    R101_3축_프론트_I_RB_PROG_ECHO_8 AT %MW84012.3 : BOOL;
    R101_3축_프론트_I_RB_SP3_8 AT %MW84013.8 : BOOL;
    R101_3축_프론트_I_RB_SP3_9 AT %MW84013.9 : BOOL;
    R101_3축_프론트_I_RB_SPARE_WORD_4 AT %MW84014 : WORD;
    R101_3축_프론트_I_RB_SP_1_12 AT %MW84011.12 : BOOL;
    R101_3축_프론트_I_RB_SP_1_13 AT %MW84011.13 : BOOL;
    R101_3축_프론트_I_RB_SP_1_14 AT %MW84011.14 : BOOL;
    R101_3축_프론트_I_RB_SP_1_15 AT %MW84011.15 : BOOL;
    R101_3축_프론트_I_RB_TC_이상 AT %MW84012.8 : BOOL;
    R101_3축_프론트_I_RB_TIP_CHANGE AT %MW84013.13 : BOOL;
    R101_3축_프론트_I_RB_TIP_DRESSING AT %MW84010.7 : BOOL;
    R101_3축_프론트_I_RB__PLT_카운터리셋완료 AT %MW84013.10 : BOOL;
    R101_3축_프론트_I_RB_공기압_이상 AT %MW84012.9 : BOOL;
    R101_3축_프론트_I_RB_냉각수_이상 AT %MW84012.10 : BOOL;
    R101_3축_프론트_I_RB_비상정지_NC AT %MW84010.8 : BOOL;
    R101_3축_프론트_I_RB_비전이상 AT %MW84012.14 : BOOL;
    R101_3축_프론트_I_RB_실러이상 AT %MW84012.13 : BOOL;
    R101_3축_프론트_I_RB_용접카운터이상 AT %MW84012.15 : BOOL;
    R101_3축_프론트_I_RB_용접타점수 AT %MW84015 : WORD;
    R101_3축_프론트_I_RB_운전준비 AT %MW84010.3 : BOOL;
    R101_3축_프론트_I_RB_원위치 AT %MW84010.0 : BOOL;
    R101_3축_프론트_I_RB_이상리셋 AT %MW84010.2 : BOOL;
    R101_3축_프론트_I_RB_자동 AT %MW84010.4 : BOOL;
    R101_3축_프론트_I_RB_자동기동 AT %MW84010.5 : BOOL;
    R101_3축_프론트_I_RB_최종_작업완료 AT %MW84010.1 : BOOL;
    R101_3축_프론트_I_RB_통신이상 AT %MW84012.12 : BOOL;
    R101_3축_프론트_M_I_RB_1차_작업완료 AT %MW20011.2 : BOOL;
    R101_3축_프론트_M_I_RB_2차_작업완료 AT %MW20011.3 : BOOL;
    R101_3축_프론트_M_I_RB_3차_작업완료 AT %MW20011.4 : BOOL;
    R101_3축_프론트_M_I_RB_4차_작업완료 AT %MW20011.5 : BOOL;
    R101_3축_프론트_M_I_RB_5차_작업완료 AT %MW20011.6 : BOOL;
    R101_3축_프론트_M_I_RB_6차_작업완료 AT %MW20011.7 : BOOL;
    R101_3축_프론트_M_I_RB_7차_작업완료 AT %MW20011.8 : BOOL;
    R101_3축_프론트_M_I_RB_PAUSE_보조 AT %MW20010.5 : BOOL;
    R101_3축_프론트_M_I_RB_PLC_RUN_CHK_이상 AT %MW20010.7 : BOOL;
    R101_3축_프론트_M_I_RB_간섭무_1 AT %MW20012.0 : BOOL;
    R101_3축_프론트_M_I_RB_간섭무_10 AT %MW20012.9 : BOOL;
    R101_3축_프론트_M_I_RB_간섭무_11 AT %MW20012.10 : BOOL;
    R101_3축_프론트_M_I_RB_간섭무_12 AT %MW20012.11 : BOOL;
    R101_3축_프론트_M_I_RB_간섭무_2 AT %MW20012.1 : BOOL;
    R101_3축_프론트_M_I_RB_간섭무_3 AT %MW20012.2 : BOOL;
    R101_3축_프론트_M_I_RB_간섭무_4 AT %MW20012.3 : BOOL;
    R101_3축_프론트_M_I_RB_간섭무_5 AT %MW20012.4 : BOOL;
    R101_3축_프론트_M_I_RB_간섭무_6 AT %MW20012.5 : BOOL;
    R101_3축_프론트_M_I_RB_간섭무_7 AT %MW20012.6 : BOOL;
    R101_3축_프론트_M_I_RB_간섭무_8 AT %MW20012.7 : BOOL;
    R101_3축_프론트_M_I_RB_간섭무_9 AT %MW20012.8 : BOOL;
    R101_3축_프론트_M_I_RB_비상정지 AT %MW20010.4 : BOOL;
    R101_3축_프론트_M_I_RB_운전준비 AT %MW20010.0 : BOOL;
    R101_3축_프론트_M_I_RB_원위치 AT %MW20010.3 : BOOL;
    R101_3축_프론트_M_I_RB_이상 AT %MW20010.2 : BOOL;
    R101_3축_프론트_M_I_RB_자동 AT %MW20010.1 : BOOL;
    R101_3축_프론트_M_I_RB_최종작업완료 AT %MW20011.0 : BOOL;
    R101_3축_프론트_M_I_RB_프로그램_이상 AT %MW20010.6 : BOOL;
    R101_3축_프론트_M_O_RB_1_CYCLE_SET AT %MW21010.3 : BOOL;
    R101_3축_프론트_M_O_RB_1_CYCLE_리셋 AT %MW21010.4 : BOOL;
    R101_3축_프론트_M_O_RB_1차_작업완료_리셋 AT %MW21012.0 : BOOL;
    R101_3축_프론트_M_O_RB_2차_작업완료_리셋 AT %MW21012.1 : BOOL;
    R101_3축_프론트_M_O_RB_2차_진입OK AT %MW21011.8 : BOOL;
    R101_3축_프론트_M_O_RB_3차_작업완료_리셋 AT %MW21012.2 : BOOL;
    R101_3축_프론트_M_O_RB_3차_진입OK AT %MW21011.9 : BOOL;
    R101_3축_프론트_M_O_RB_4차_작업완료_리셋 AT %MW21012.3 : BOOL;
    R101_3축_프론트_M_O_RB_4차_진입OK AT %MW21011.10 : BOOL;
    R101_3축_프론트_M_O_RB_5차_작업완료_리셋 AT %MW21012.4 : BOOL;
    R101_3축_프론트_M_O_RB_5차_진입OK AT %MW21011.11 : BOOL;
    R101_3축_프론트_M_O_RB_6차_작업완료_리셋 AT %MW21012.5 : BOOL;
    R101_3축_프론트_M_O_RB_6차_진입OK AT %MW21011.12 : BOOL;
    R101_3축_프론트_M_O_RB_7차_작업완료_리셋 AT %MW21012.6 : BOOL;
    R101_3축_프론트_M_O_RB_7차_진입OK AT %MW21011.13 : BOOL;
    R101_3축_프론트_M_O_RB_ATD_OK AT %MW21010.6 : BOOL;
    R101_3축_프론트_M_O_RB_PLT_10_진입OK AT %MW21013.10 : BOOL;
    R101_3축_프론트_M_O_RB_PLT_11_진입OK AT %MW21013.11 : BOOL;
    R101_3축_프론트_M_O_RB_PLT_12_진입OK AT %MW21013.12 : BOOL;
    R101_3축_프론트_M_O_RB_PLT_1_진입OK AT %MW21013.1 : BOOL;
    R101_3축_프론트_M_O_RB_PLT_2_진입OK AT %MW21013.2 : BOOL;
    R101_3축_프론트_M_O_RB_PLT_3_진입OK AT %MW21013.3 : BOOL;
    R101_3축_프론트_M_O_RB_PLT_4_진입OK AT %MW21013.4 : BOOL;
    R101_3축_프론트_M_O_RB_PLT_5_진입OK AT %MW21013.5 : BOOL;
    R101_3축_프론트_M_O_RB_PLT_6_진입OK AT %MW21013.6 : BOOL;
    R101_3축_프론트_M_O_RB_PLT_7_진입OK AT %MW21013.7 : BOOL;
    R101_3축_프론트_M_O_RB_PLT_8_진입OK AT %MW21013.8 : BOOL;
    R101_3축_프론트_M_O_RB_PLT_9_진입OK AT %MW21013.9 : BOOL;
    R101_3축_프론트_M_O_RB_PLT_카운터리셋_보조 AT %MW21010.10 : BOOL;
    R101_3축_프론트_M_O_RB_RESTART_OK AT %MW21010.2 : BOOL;
    R101_3축_프론트_M_O_RB_START_OK AT %MW21010.0 : BOOL;
    R101_3축_프론트_M_O_RB_TEST_MODE_5000회 AT %MW21010.12 : BOOL;
    R101_3축_프론트_M_O_RB_TIP_교체_시작 AT %MW21010.7 : BOOL;
    R101_3축_프론트_M_O_RB_TIP_교체_완료 AT %MW21010.8 : BOOL;
    R101_3축_프론트_M_O_RB_VIP_MODE AT %MW21010.11 : BOOL;
    R101_3축_프론트_M_O_RB_냉각수_차단_요청 AT %MW21010.9 : BOOL;
    R101_3축_프론트_M_O_RB_진입OK_AX차종 AT %MW21011.0 : BOOL;
    R101_3축_프론트_M_O_RB_진입OK_B차종 AT %MW21011.1 : BOOL;
    R101_3축_프론트_M_O_RB_진입OK_C차종 AT %MW21011.2 : BOOL;
    R101_3축_프론트_M_O_RB_진입OK_D차종 AT %MW21011.3 : BOOL;
    R101_3축_프론트_M_O_RB_진입OK_E차종 AT %MW21011.4 : BOOL;
    R101_3축_프론트_M_O_RB_진입OK_F차종 AT %MW21011.5 : BOOL;
    R101_3축_프론트_M_O_RB_진입OK_G차종 AT %MW21011.6 : BOOL;
    R101_3축_프론트_M_O_RB_진입OK_H차종 AT %MW21011.7 : BOOL;
    R101_3축_프론트_M_O_RB_최종_작업완료_리셋 AT %MW21010.5 : BOOL;
    R101_3축_프론트_M_O_RB_프로그램_OK AT %MW21010.1 : BOOL;
    R101_3축_프론트_M_RB_PROG_NO AT %MW20014 : WORD;
    R101_3축_프론트_O_RB_0_5S_통신_CHK AT %MW94013.14 : BOOL;
    R101_3축_프론트_O_RB_2차_진입OK AT %MW94011.8 : BOOL;
    R101_3축_프론트_O_RB_3차_진입OK AT %MW94011.9 : BOOL;
    R101_3축_프론트_O_RB_4차_진입OK AT %MW94011.10 : BOOL;
    R101_3축_프론트_O_RB_5차_진입OK AT %MW94011.11 : BOOL;
    R101_3축_프론트_O_RB_6차_진입OK AT %MW94011.12 : BOOL;
    R101_3축_프론트_O_RB_7차_진입OK AT %MW94011.13 : BOOL;
    R101_3축_프론트_O_RB_AX_1차_진입OK AT %MW94011.0 : BOOL;
    R101_3축_프론트_O_RB_B_1차_진입OK AT %MW94011.1 : BOOL;
    R101_3축_프론트_O_RB_C_1차_진입OK AT %MW94011.2 : BOOL;
    R101_3축_프론트_O_RB_D_1차_진입OK AT %MW94011.3 : BOOL;
    R101_3축_프론트_O_RB_EACH_작업완료_리셋 AT %MW94010.14 : BOOL;
    R101_3축_프론트_O_RB_EXT_READY AT %MW94010.11 : BOOL;
    R101_3축_프론트_O_RB_E_1차_진입OK AT %MW94011.4 : BOOL;
    R101_3축_프론트_O_RB_F_1차_진입OK AT %MW94011.5 : BOOL;
    R101_3축_프론트_O_RB_GATE_OPEN_NC AT %MW94013.11 : BOOL;
    R101_3축_프론트_O_RB_G_1차_진입OK AT %MW94011.6 : BOOL;
    R101_3축_프론트_O_RB_H_1차_진입OK AT %MW94011.7 : BOOL;
    R101_3축_프론트_O_RB_MUTUAL_INT1 AT %MW94013.0 : BOOL;
    R101_3축_프론트_O_RB_MUTUAL_INT2 AT %MW94013.1 : BOOL;
    R101_3축_프론트_O_RB_MUTUAL_INT3 AT %MW94013.2 : BOOL;
    R101_3축_프론트_O_RB_MUTUAL_INT4 AT %MW94013.3 : BOOL;
    R101_3축_프론트_O_RB_MUTUAL_INT5 AT %MW94013.4 : BOOL;
    R101_3축_프론트_O_RB_MUTUAL_INT6 AT %MW94013.5 : BOOL;
    R101_3축_프론트_O_RB_MUTUAL_INT7 AT %MW94013.6 : BOOL;
    R101_3축_프론트_O_RB_MUTUAL_INT8 AT %MW94013.7 : BOOL;
    R101_3축_프론트_O_RB_OUTPUT AT %MW94010 : ARRAY[0..3] OF WORD;
    R101_3축_프론트_O_RB_PAUSE_NC AT %MW94010.13 : BOOL;
    R101_3축_프론트_O_RB_PLT10_진입OK AT %MW94012.9 : BOOL;
    R101_3축_프론트_O_RB_PLT11_진입OK AT %MW94012.10 : BOOL;
    R101_3축_프론트_O_RB_PLT12_진입OK AT %MW94012.11 : BOOL;
    R101_3축_프론트_O_RB_PLT1_진입OK AT %MW94012.0 : BOOL;
    R101_3축_프론트_O_RB_PLT2_진입OK AT %MW94012.1 : BOOL;
    R101_3축_프론트_O_RB_PLT3_진입OK AT %MW94012.2 : BOOL;
    R101_3축_프론트_O_RB_PLT4_진입OK AT %MW94012.3 : BOOL;
    R101_3축_프론트_O_RB_PLT5_진입OK AT %MW94012.4 : BOOL;
    R101_3축_프론트_O_RB_PLT6_진입OK AT %MW94012.5 : BOOL;
    R101_3축_프론트_O_RB_PLT7_진입OK AT %MW94012.6 : BOOL;
    R101_3축_프론트_O_RB_PLT8_진입OK AT %MW94012.7 : BOOL;
    R101_3축_프론트_O_RB_PLT9_진입OK AT %MW94012.8 : BOOL;
    R101_3축_프론트_O_RB_PLT_COUNT_리셋_COND AT %MW94013.10 : BOOL;
    R101_3축_프론트_O_RB_PROG_선택1 AT %MW94010.0 : BOOL;
    R101_3축_프론트_O_RB_PROG_선택128 AT %MW94010.7 : BOOL;
    R101_3축_프론트_O_RB_PROG_선택16 AT %MW94010.4 : BOOL;
    R101_3축_프론트_O_RB_PROG_선택2 AT %MW94010.1 : BOOL;
    R101_3축_프론트_O_RB_PROG_선택32 AT %MW94010.5 : BOOL;
    R101_3축_프론트_O_RB_PROG_선택4 AT %MW94010.2 : BOOL;
    R101_3축_프론트_O_RB_PROG_선택64 AT %MW94010.6 : BOOL;
    R101_3축_프론트_O_RB_PROG_선택8 AT %MW94010.3 : BOOL;
    R101_3축_프론트_O_RB_SP_1_14 AT %MW94011.14 : BOOL;
    R101_3축_프론트_O_RB_SP_1_15 AT %MW94011.15 : BOOL;
    R101_3축_프론트_O_RB_SP_2_12 AT %MW94012.12 : BOOL;
    R101_3축_프론트_O_RB_SP_2_13 AT %MW94012.13 : BOOL;
    R101_3축_프론트_O_RB_SP_2_14 AT %MW94012.14 : BOOL;
    R101_3축_프론트_O_RB_SP_5000TH_ON AT %MW94012.15 : BOOL;
    R101_3축_프론트_O_RB_TIP_CHANGE_END AT %MW94013.9 : BOOL;
    R101_3축_프론트_O_RB_TIP_CHANGE_START AT %MW94013.8 : BOOL;
    R101_3축_프론트_O_RB_TIP_DRESS_SATRT AT %MW94010.12 : BOOL;
    R101_3축_프론트_O_RB_VIP_MODE AT %MW94013.15 : BOOL;
    R101_3축_프론트_O_RB_기동 AT %MW94010.9 : BOOL;
    R101_3축_프론트_O_RB_냉각수차단 AT %MW94010.15 : BOOL;
    R101_3축_프론트_O_RB_부저정지 AT %MW94013.13 : BOOL;
    R101_3축_프론트_O_RB_비상정지_NC AT %MW94013.12 : BOOL;
    R101_3축_프론트_O_RB_이상_리셋 AT %MW94010.10 : BOOL;
    R101_3축_프론트_O_RB_작업완료_리셋 AT %MW94010.8 : BOOL;
    R102_1_1_I_RB_0_5_COMM_CHK AT %MW84093.14 : BOOL;
    R102_1_1_I_RB_10차_간섭무 AT %MW84091.9 : BOOL;
    R102_1_1_I_RB_11차_간섭무 AT %MW84091.10 : BOOL;
    R102_1_1_I_RB_12차_간섭무 AT %MW84091.11 : BOOL;
    R102_1_1_I_RB_1차_간섭무 AT %MW84091.0 : BOOL;
    R102_1_1_I_RB_1차_작업완료 AT %MW84090.9 : BOOL;
    R102_1_1_I_RB_2차_간섭무 AT %MW84091.1 : BOOL;
    R102_1_1_I_RB_2차_작업완료 AT %MW84090.10 : BOOL;
    R102_1_1_I_RB_3차_간섭무 AT %MW84091.2 : BOOL;
    R102_1_1_I_RB_3차_작업완료 AT %MW84090.11 : BOOL;
    R102_1_1_I_RB_4차_간섭무 AT %MW84091.3 : BOOL;
    R102_1_1_I_RB_4차_작업완료 AT %MW84090.12 : BOOL;
    R102_1_1_I_RB_5차_간섭무 AT %MW84091.4 : BOOL;
    R102_1_1_I_RB_5차_작업완료 AT %MW84090.13 : BOOL;
    R102_1_1_I_RB_6차_간섭무 AT %MW84091.5 : BOOL;
    R102_1_1_I_RB_6차_작업완료 AT %MW84090.14 : BOOL;
    R102_1_1_I_RB_7차_간섭무 AT %MW84091.6 : BOOL;
    R102_1_1_I_RB_7차_작업완료 AT %MW84090.15 : BOOL;
    R102_1_1_I_RB_8차_간섭무 AT %MW84091.7 : BOOL;
    R102_1_1_I_RB_9차_간섭무 AT %MW84091.8 : BOOL;
    R102_1_1_I_RB_AB_NORMAL_선택 AT %MW84090.6 : BOOL;
    R102_1_1_I_RB_GUN1_FIXED_TIP AT %MW84097 : WORD;
    R102_1_1_I_RB_GUN1_MOVING_TIP AT %MW84096 : WORD;
    R102_1_1_I_RB_GUN2_FIXED_TIP AT %MW84099 : WORD;
    R102_1_1_I_RB_GUN2_MOVING_TIP AT %MW84098 : WORD;
    R102_1_1_I_RB_INPUT AT %MW84090 : ARRAY[0..3] OF WORD;
    R102_1_1_I_RB_LS_이상 AT %MW84092.11 : BOOL;
    R102_1_1_I_RB_MOTOR_MC_ON AT %MW84093.15 : BOOL;
    R102_1_1_I_RB_MUTUAL_INT1 AT %MW84093.0 : BOOL;
    R102_1_1_I_RB_MUTUAL_INT2 AT %MW84093.1 : BOOL;
    R102_1_1_I_RB_MUTUAL_INT3 AT %MW84093.2 : BOOL;
    R102_1_1_I_RB_MUTUAL_INT4 AT %MW84093.3 : BOOL;
    R102_1_1_I_RB_MUTUAL_INT5 AT %MW84093.4 : BOOL;
    R102_1_1_I_RB_MUTUAL_INT6 AT %MW84093.5 : BOOL;
    R102_1_1_I_RB_MUTUAL_INT7 AT %MW84093.6 : BOOL;
    R102_1_1_I_RB_MUTUAL_INT8 AT %MW84093.7 : BOOL;
    R102_1_1_I_RB_PLT_UNLOAD_완료 AT %MW84093.11 : BOOL;
    R102_1_1_I_RB_PLT_최종UNLOAD_완료 AT %MW84093.12 : BOOL;
    R102_1_1_I_RB_PROG_ECHO_1 AT %MW84092.0 : BOOL;
    R102_1_1_I_RB_PROG_ECHO_128 AT %MW84092.7 : BOOL;
    R102_1_1_I_RB_PROG_ECHO_16 AT %MW84092.4 : BOOL;
    R102_1_1_I_RB_PROG_ECHO_2 AT %MW84092.1 : BOOL;
    R102_1_1_I_RB_PROG_ECHO_32 AT %MW84092.5 : BOOL;
    R102_1_1_I_RB_PROG_ECHO_4 AT %MW84092.2 : BOOL;
    R102_1_1_I_RB_PROG_ECHO_64 AT %MW84092.6 : BOOL;
    R102_1_1_I_RB_PROG_ECHO_8 AT %MW84092.3 : BOOL;
    R102_1_1_I_RB_SP3_8 AT %MW84093.8 : BOOL;
    R102_1_1_I_RB_SP3_9 AT %MW84093.9 : BOOL;
    R102_1_1_I_RB_SPARE_WORD_4 AT %MW84094 : WORD;
    R102_1_1_I_RB_SP_1_12 AT %MW84091.12 : BOOL;
    R102_1_1_I_RB_SP_1_13 AT %MW84091.13 : BOOL;
    R102_1_1_I_RB_SP_1_14 AT %MW84091.14 : BOOL;
    R102_1_1_I_RB_SP_1_15 AT %MW84091.15 : BOOL;
    R102_1_1_I_RB_TC_이상 AT %MW84092.8 : BOOL;
    R102_1_1_I_RB_TIP_CHANGE AT %MW84093.13 : BOOL;
    R102_1_1_I_RB_TIP_DRESSING AT %MW84090.7 : BOOL;
    R102_1_1_I_RB__PLT_카운터리셋완료 AT %MW84093.10 : BOOL;
    R102_1_1_I_RB_공기압_이상 AT %MW84092.9 : BOOL;
    R102_1_1_I_RB_냉각수_이상 AT %MW84092.10 : BOOL;
    R102_1_1_I_RB_비상정지_NC AT %MW84090.8 : BOOL;
    R102_1_1_I_RB_비전이상 AT %MW84092.14 : BOOL;
    R102_1_1_I_RB_실러이상 AT %MW84092.13 : BOOL;
    R102_1_1_I_RB_용접카운터이상 AT %MW84092.15 : BOOL;
    R102_1_1_I_RB_용접타점수 AT %MW84095 : WORD;
    R102_1_1_I_RB_운전준비 AT %MW84090.3 : BOOL;
    R102_1_1_I_RB_원위치 AT %MW84090.0 : BOOL;
    R102_1_1_I_RB_이상리셋 AT %MW84090.2 : BOOL;
    R102_1_1_I_RB_자동 AT %MW84090.4 : BOOL;
    R102_1_1_I_RB_자동기동 AT %MW84090.5 : BOOL;
    R102_1_1_I_RB_최종_작업완료 AT %MW84090.1 : BOOL;
    R102_1_1_I_RB_통신이상 AT %MW84092.12 : BOOL;
    R102_1_1_M_DATA_삭제_PLS AT %MW9002.0 : BOOL; (* R102_1_1_M_DATA_삭제_PLS *)
    R102_1_1_M_DATA_삭제_SIGN AT %MW9002.1 : BOOL; (* R102_1_1_M_DATA_삭제_SIGN *)
    R102_1_1_M_DATA_삭제_완료 AT %MW9002.2 : BOOL; (* R102_1_1_M_DATA_삭제_완료 *)
    R102_1_1_M_DATA_전송_MEMO AT %MW9002.8 : BOOL; (* R102_1_1_M_DATA_전송_MEMO *)
    R102_1_1_M_DATA_전송_PLS AT %MW9002.9 : BOOL; (* R102_1_1_M_DATA_전송_PLS *)
    R102_1_1_M_DATA_전송_SIGN AT %MW9002.10 : BOOL; (* R102_1_1_M_DATA_전송_SIGN *)
    R102_1_1_M_DATA_전송_완료 AT %MW9002.11 : BOOL; (* R102_1_1_M_DATA_전송_완료 *)
    R102_1_1_M_I_RB_1차_작업완료 AT %MW20091.2 : BOOL;
    R102_1_1_M_I_RB_2차_작업완료 AT %MW20091.3 : BOOL;
    R102_1_1_M_I_RB_3차_작업완료 AT %MW20091.4 : BOOL;
    R102_1_1_M_I_RB_4차_작업완료 AT %MW20091.5 : BOOL;
    R102_1_1_M_I_RB_5차_작업완료 AT %MW20091.6 : BOOL;
    R102_1_1_M_I_RB_6차_작업완료 AT %MW20091.7 : BOOL;
    R102_1_1_M_I_RB_7차_작업완료 AT %MW20091.8 : BOOL;
    R102_1_1_M_I_RB_PAUSE_보조 AT %MW20090.5 : BOOL;
    R102_1_1_M_I_RB_PLC_RUN_CHK_이상 AT %MW20090.7 : BOOL;
    R102_1_1_M_I_RB_간섭무_1 AT %MW20092.0 : BOOL;
    R102_1_1_M_I_RB_간섭무_10 AT %MW20092.9 : BOOL;
    R102_1_1_M_I_RB_간섭무_11 AT %MW20092.10 : BOOL;
    R102_1_1_M_I_RB_간섭무_12 AT %MW20092.11 : BOOL;
    R102_1_1_M_I_RB_간섭무_2 AT %MW20092.1 : BOOL;
    R102_1_1_M_I_RB_간섭무_3 AT %MW20092.2 : BOOL;
    R102_1_1_M_I_RB_간섭무_4 AT %MW20092.3 : BOOL;
    R102_1_1_M_I_RB_간섭무_5 AT %MW20092.4 : BOOL;
    R102_1_1_M_I_RB_간섭무_6 AT %MW20092.5 : BOOL;
    R102_1_1_M_I_RB_간섭무_7 AT %MW20092.6 : BOOL;
    R102_1_1_M_I_RB_간섭무_8 AT %MW20092.7 : BOOL;
    R102_1_1_M_I_RB_간섭무_9 AT %MW20092.8 : BOOL;
    R102_1_1_M_I_RB_비상정지 AT %MW20090.4 : BOOL;
    R102_1_1_M_I_RB_운전준비 AT %MW20090.0 : BOOL;
    R102_1_1_M_I_RB_원위치 AT %MW20090.3 : BOOL;
    R102_1_1_M_I_RB_이상 AT %MW20090.2 : BOOL;
    R102_1_1_M_I_RB_자동 AT %MW20090.1 : BOOL;
    R102_1_1_M_I_RB_최종작업완료 AT %MW20091.0 : BOOL;
    R102_1_1_M_I_RB_프로그램_이상 AT %MW20090.6 : BOOL;
    R102_1_1_M_O_RB_1_CYCLE_SET AT %MW21090.3 : BOOL;
    R102_1_1_M_O_RB_1_CYCLE_리셋 AT %MW21090.4 : BOOL;
    R102_1_1_M_O_RB_1차_작업완료_리셋 AT %MW21092.0 : BOOL;
    R102_1_1_M_O_RB_2차_작업완료_리셋 AT %MW21092.1 : BOOL;
    R102_1_1_M_O_RB_2차_진입OK AT %MW21091.8 : BOOL;
    R102_1_1_M_O_RB_3차_작업완료_리셋 AT %MW21092.2 : BOOL;
    R102_1_1_M_O_RB_3차_진입OK AT %MW21091.9 : BOOL;
    R102_1_1_M_O_RB_4차_작업완료_리셋 AT %MW21092.3 : BOOL;
    R102_1_1_M_O_RB_4차_진입OK AT %MW21091.10 : BOOL;
    R102_1_1_M_O_RB_5차_작업완료_리셋 AT %MW21092.4 : BOOL;
    R102_1_1_M_O_RB_5차_진입OK AT %MW21091.11 : BOOL;
    R102_1_1_M_O_RB_6차_작업완료_리셋 AT %MW21092.5 : BOOL;
    R102_1_1_M_O_RB_6차_진입OK AT %MW21091.12 : BOOL;
    R102_1_1_M_O_RB_7차_작업완료_리셋 AT %MW21092.6 : BOOL;
    R102_1_1_M_O_RB_7차_진입OK AT %MW21091.13 : BOOL;
    R102_1_1_M_O_RB_ATD_OK AT %MW21090.6 : BOOL;
    R102_1_1_M_O_RB_PLT_10_진입OK AT %MW21093.10 : BOOL;
    R102_1_1_M_O_RB_PLT_11_진입OK AT %MW21093.11 : BOOL;
    R102_1_1_M_O_RB_PLT_12_진입OK AT %MW21093.12 : BOOL;
    R102_1_1_M_O_RB_PLT_1_진입OK AT %MW21093.1 : BOOL;
    R102_1_1_M_O_RB_PLT_2_진입OK AT %MW21093.2 : BOOL;
    R102_1_1_M_O_RB_PLT_3_진입OK AT %MW21093.3 : BOOL;
    R102_1_1_M_O_RB_PLT_4_진입OK AT %MW21093.4 : BOOL;
    R102_1_1_M_O_RB_PLT_5_진입OK AT %MW21093.5 : BOOL;
    R102_1_1_M_O_RB_PLT_6_진입OK AT %MW21093.6 : BOOL;
    R102_1_1_M_O_RB_PLT_7_진입OK AT %MW21093.7 : BOOL;
    R102_1_1_M_O_RB_PLT_8_진입OK AT %MW21093.8 : BOOL;
    R102_1_1_M_O_RB_PLT_9_진입OK AT %MW21093.9 : BOOL;
    R102_1_1_M_O_RB_PLT_카운터리셋_보조 AT %MW21090.10 : BOOL;
    R102_1_1_M_O_RB_RESTART_OK AT %MW21090.2 : BOOL;
    R102_1_1_M_O_RB_START_OK AT %MW21090.0 : BOOL;
    R102_1_1_M_O_RB_TEST_MODE_5000회 AT %MW21090.12 : BOOL;
    R102_1_1_M_O_RB_TIP_교체_시작 AT %MW21090.7 : BOOL;
    R102_1_1_M_O_RB_TIP_교체_완료 AT %MW21090.8 : BOOL;
    R102_1_1_M_O_RB_VIP_MODE AT %MW21090.11 : BOOL;
    R102_1_1_M_O_RB_냉각수_차단_요청 AT %MW21090.9 : BOOL;
    R102_1_1_M_O_RB_진입OK_AX차종 AT %MW21091.0 : BOOL;
    R102_1_1_M_O_RB_진입OK_B차종 AT %MW21091.1 : BOOL;
    R102_1_1_M_O_RB_진입OK_C차종 AT %MW21091.2 : BOOL;
    R102_1_1_M_O_RB_진입OK_D차종 AT %MW21091.3 : BOOL;
    R102_1_1_M_O_RB_진입OK_E차종 AT %MW21091.4 : BOOL;
    R102_1_1_M_O_RB_진입OK_F차종 AT %MW21091.5 : BOOL;
    R102_1_1_M_O_RB_진입OK_G차종 AT %MW21091.6 : BOOL;
    R102_1_1_M_O_RB_진입OK_H차종 AT %MW21091.7 : BOOL;
    R102_1_1_M_O_RB_최종_작업완료_리셋 AT %MW21090.5 : BOOL;
    R102_1_1_M_O_RB_프로그램_OK AT %MW21090.1 : BOOL;
    R102_1_1_M_RB_PROG_NO AT %MW20094 : WORD;
    R102_1_1_M_RB_통신이상 AT %MW1524.3 : BOOL;
    R102_1_1_M_SEQ AT %MW10040 : WORD; (* R102_1_1_M_SEQ *)
    R102_1_1_M_STN_차종_NONE AT %MW1502.3 : BOOL;
    R102_1_1_M_STN_차종_ON AT %MW1502.2 : BOOL;
    R102_1_1_M_VIN_NO_1_2 AT %MW10051 : WORD; (* R102_1_1_M_VIN_NO_1_2 *)
    R102_1_1_M_VIN_NO_3_4 AT %MW10052 : WORD; (* R102_1_1_M_VIN_NO_3_4 *)
    R102_1_1_M_VIN_NO_5_6 AT %MW10053 : WORD; (* R102_1_1_M_VIN_NO_5_6 *)
    R102_1_1_M_VIN_NO_7_8 AT %MW10054 : WORD; (* R102_1_1_M_VIN_NO_7_8 *)
    R102_1_1_M_VIN_NO_9_10 AT %MW10055 : WORD; (* R102_1_1_M_VIN_NO_9_10 *)
    R102_1_1_M_차종1_AX AT %MW10041.0 : BOOL; (* R102_1_1_M_차종1_AX *)
    R102_1_1_M_차종1_B AT %MW10041.1 : BOOL; (* R102_1_1_M_차종1_B *)
    R102_1_1_M_차종1_C AT %MW10041.2 : BOOL; (* R102_1_1_M_차종1_C *)
    R102_1_1_M_차종1_D AT %MW10041.3 : BOOL; (* R102_1_1_M_차종1_D *)
    R102_1_1_M_차종1_E AT %MW10041.4 : BOOL; (* R102_1_1_M_차종1_E *)
    R102_1_1_M_차종1_F AT %MW10041.5 : BOOL; (* R102_1_1_M_차종1_F *)
    R102_1_1_M_차종1_G AT %MW10041.6 : BOOL; (* R102_1_1_M_차종1_G *)
    R102_1_1_M_차종1_H AT %MW10041.7 : BOOL; (* R102_1_1_M_차종1_H *)
    R102_1_1_M_차종2_3DR AT %MW10041.8 : BOOL; (* R102_1_1_M_차종2_3DR *)
    R102_1_1_M_차종2_4DR AT %MW10041.9 : BOOL; (* R102_1_1_M_차종2_4DR *)
    R102_1_1_M_차종2_5DR AT %MW10041.10 : BOOL; (* R102_1_1_M_차종2_5DR *)
    R102_1_1_M_차종2_SP1 AT %MW10041.12 : BOOL; (* R102_1_1_M_차종2_SP1 *)
    R102_1_1_M_차종2_SP2 AT %MW10041.13 : BOOL; (* R102_1_1_M_차종2_SP2 *)
    R102_1_1_M_차종2_WGN AT %MW10041.11 : BOOL; (* R102_1_1_M_차종2_WGN *)
    R102_1_1_M_차종3_LHD AT %MW10041.14 : BOOL; (* R102_1_1_M_차종3_LHD *)
    R102_1_1_M_차종3_RHD AT %MW10041.15 : BOOL; (* R102_1_1_M_차종3_RHD *)
    R102_1_1_M_차종4_EEC AT %MW10042.3 : BOOL; (* R102_1_1_M_차종4_EEC *)
    R102_1_1_M_차종4_SP1 AT %MW10042.8 : BOOL; (* R102_1_1_M_차종4_SP1 *)
    R102_1_1_M_차종4_SP2 AT %MW10042.9 : BOOL; (* R102_1_1_M_차종4_SP2 *)
    R102_1_1_M_차종4_SP3 AT %MW10042.11 : BOOL; (* R102_1_1_M_차종4_SP3 *)
    R102_1_1_M_차종4_SP4 AT %MW10042.12 : BOOL; (* R102_1_1_M_차종4_SP4 *)
    R102_1_1_M_차종4_SP5 AT %MW10042.13 : BOOL; (* R102_1_1_M_차종4_SP5 *)
    R102_1_1_M_차종4_SP6 AT %MW10042.14 : BOOL; (* R102_1_1_M_차종4_SP6 *)
    R102_1_1_M_차종4_SP7 AT %MW10042.15 : BOOL; (* R102_1_1_M_차종4_SP7 *)
    R102_1_1_M_차종4_내수 AT %MW10042.0 : BOOL; (* R102_1_1_M_차종4_내수 *)
    R102_1_1_M_차종4_러시아 AT %MW10042.10 : BOOL; (* R102_1_1_M_차종4_러시아 *)
    R102_1_1_M_차종4_북미 AT %MW10042.2 : BOOL; (* R102_1_1_M_차종4_북미 *)
    R102_1_1_M_차종4_브라질 AT %MW10042.7 : BOOL; (* R102_1_1_M_차종4_브라질 *)
    R102_1_1_M_차종4_수출 AT %MW10042.1 : BOOL; (* R102_1_1_M_차종4_수출 *)
    R102_1_1_M_차종4_중국 AT %MW10042.6 : BOOL; (* R102_1_1_M_차종4_중국 *)
    R102_1_1_M_차종4_중동 AT %MW10042.5 : BOOL; (* R102_1_1_M_차종4_중동 *)
    R102_1_1_M_차종4_호주 AT %MW10042.4 : BOOL; (* R102_1_1_M_차종4_호주 *)
    R102_1_1_M_차종5_AT AT %MW10043.1 : BOOL; (* R102_1_1_M_차종5_AT *)
    R102_1_1_M_차종5_MT AT %MW10043.0 : BOOL; (* R102_1_1_M_차종5_MT *)
    R102_1_1_M_차종5_SP1 AT %MW10043.2 : BOOL; (* R102_1_1_M_차종5_SP1 *)
    R102_1_1_M_차종6_DSROOF AT %MW10043.6 : BOOL; (* R102_1_1_M_차종6_DSROOF *)
    R102_1_1_M_차종6_SP1 AT %MW10043.7 : BOOL; (* R102_1_1_M_차종6_SP1 *)
    R102_1_1_M_차종6_썬루프 AT %MW10043.4 : BOOL; (* R102_1_1_M_차종6_썬루프 *)
    R102_1_1_M_차종6_일반루프 AT %MW10043.3 : BOOL; (* R102_1_1_M_차종6_일반루프 *)
    R102_1_1_M_차종6_파노라마루프 AT %MW10043.5 : BOOL; (* R102_1_1_M_차종6_파노라마루프 *)
    R102_1_1_M_차종7_DSL AT %MW10043.9 : BOOL; (* R102_1_1_M_차종7_DSL *)
    R102_1_1_M_차종7_GSL AT %MW10043.8 : BOOL; (* R102_1_1_M_차종7_GSL *)
    R102_1_1_M_차종7_SP1 AT %MW10043.10 : BOOL; (* R102_1_1_M_차종7_SP1 *)
    R102_1_1_M_차종7_SP2 AT %MW10043.11 : BOOL; (* R102_1_1_M_차종7_SP2 *)
    R102_1_1_M_차종7_SP3 AT %MW10043.12 : BOOL; (* R102_1_1_M_차종7_SP3 *)
    R102_1_1_M_차종7_SP4 AT %MW10043.13 : BOOL; (* R102_1_1_M_차종7_SP4 *)
    R102_1_1_M_차종7_SP5 AT %MW10043.14 : BOOL; (* R102_1_1_M_차종7_SP5 *)
    R102_1_1_M_차종7_SP6 AT %MW10043.15 : BOOL; (* R102_1_1_M_차종7_SP6 *)
    R102_1_1_M_차종8_2WD AT %MW10044.0 : BOOL; (* R102_1_1_M_차종8_2WD *)
    R102_1_1_M_차종8_4WD AT %MW10044.1 : BOOL; (* R102_1_1_M_차종8_4WD *)
    R102_1_1_M_차종8_SP1 AT %MW10044.2 : BOOL; (* R102_1_1_M_차종8_SP1 *)
    R102_1_1_M_차종9_MPI AT %MW10044.3 : BOOL; (* R102_1_1_M_차종9_MPI *)
    R102_1_1_M_차종9_SP1 AT %MW10044.5 : BOOL; (* R102_1_1_M_차종9_SP1 *)
    R102_1_1_M_차종9_SP10 AT %MW10044.14 : BOOL; (* R102_1_1_M_차종9_SP10 *)
    R102_1_1_M_차종9_SP11 AT %MW10044.15 : BOOL; (* R102_1_1_M_차종9_SP11 *)
    R102_1_1_M_차종9_SP2 AT %MW10044.6 : BOOL; (* R102_1_1_M_차종9_SP2 *)
    R102_1_1_M_차종9_SP3 AT %MW10044.7 : BOOL; (* R102_1_1_M_차종9_SP3 *)
    R102_1_1_M_차종9_SP4 AT %MW10044.8 : BOOL; (* R102_1_1_M_차종9_SP4 *)
    R102_1_1_M_차종9_SP5 AT %MW10044.9 : BOOL; (* R102_1_1_M_차종9_SP5 *)
    R102_1_1_M_차종9_SP6 AT %MW10044.10 : BOOL; (* R102_1_1_M_차종9_SP6 *)
    R102_1_1_M_차종9_SP7 AT %MW10044.11 : BOOL; (* R102_1_1_M_차종9_SP7 *)
    R102_1_1_M_차종9_SP8 AT %MW10044.12 : BOOL; (* R102_1_1_M_차종9_SP8 *)
    R102_1_1_M_차종9_SP9 AT %MW10044.13 : BOOL; (* R102_1_1_M_차종9_SP9 *)
    R102_1_1_M_차종9_T_GDI AT %MW10044.4 : BOOL; (* R102_1_1_M_차종9_T_GDI *)
    R102_1_1_M_차종_AS AT %MW10050.9 : BOOL; (* R102_1_1_M_차종_AS *)
    R102_1_1_M_차종_OPT1_R_RACK_무 AT %MW10045.3 : BOOL; (* R102_1_1_M_차종_OPT1_R_RACK_무 *)
    R102_1_1_M_차종_OPT1_R_RACK_유 AT %MW10045.2 : BOOL; (* R102_1_1_M_차종_OPT1_R_RACK_유 *)
    R102_1_1_M_차종_OPT1_SP1 AT %MW10045.10 : BOOL; (* R102_1_1_M_차종_OPT1_SP1 *)
    R102_1_1_M_차종_OPT1_SP2 AT %MW10045.11 : BOOL; (* R102_1_1_M_차종_OPT1_SP2 *)
    R102_1_1_M_차종_OPT1_SP3 AT %MW10045.12 : BOOL; (* R102_1_1_M_차종_OPT1_SP3 *)
    R102_1_1_M_차종_OPT1_SP4 AT %MW10045.13 : BOOL; (* R102_1_1_M_차종_OPT1_SP4 *)
    R102_1_1_M_차종_OPT1_SP5 AT %MW10045.14 : BOOL; (* R102_1_1_M_차종_OPT1_SP5 *)
    R102_1_1_M_차종_OPT1_SP6 AT %MW10045.15 : BOOL; (* R102_1_1_M_차종_OPT1_SP6 *)
    R102_1_1_M_차종_OPT1_S_REP_EATER_무 AT %MW10045.7 : BOOL; (* R102_1_1_M_차종_OPT1_S_REP_EATER_무 *)
    R102_1_1_M_차종_OPT1_S_REP_EATER_유 AT %MW10045.6 : BOOL; (* R102_1_1_M_차종_OPT1_S_REP_EATER_유 *)
    R102_1_1_M_차종_OPT1_VAN_무 AT %MW10045.9 : BOOL; (* R102_1_1_M_차종_OPT1_VAN_무 *)
    R102_1_1_M_차종_OPT1_VAN_유 AT %MW10045.8 : BOOL; (* R102_1_1_M_차종_OPT1_VAN_유 *)
    R102_1_1_M_차종_OPT1_슬라이딩_무 AT %MW10045.1 : BOOL; (* R102_1_1_M_차종_OPT1_슬라이딩_무 *)
    R102_1_1_M_차종_OPT1_슬라이딩_유 AT %MW10045.0 : BOOL; (* R102_1_1_M_차종_OPT1_슬라이딩_유 *)
    R102_1_1_M_차종_OPT1_폴딩_무 AT %MW10045.5 : BOOL; (* R102_1_1_M_차종_OPT1_폴딩_무 *)
    R102_1_1_M_차종_OPT1_폴딩_유 AT %MW10045.4 : BOOL; (* R102_1_1_M_차종_OPT1_폴딩_유 *)
    R102_1_1_M_차종_OPT2_SP_WORD1 AT %MW10046 : WORD; (* R102_1_1_M_차종_OPT2_SP_WORD1 *)
    R102_1_1_M_차종_OPT3_SP_WORD2 AT %MW10047 : WORD; (* R102_1_1_M_차종_OPT3_SP_WORD2 *)
    R102_1_1_M_차종_OPT4_SP_WORD3 AT %MW10048 : WORD; (* R102_1_1_M_차종_OPT4_SP_WORD3 *)
    R102_1_1_M_차종_OPT5_SP_WORD4 AT %MW10049 : WORD; (* R102_1_1_M_차종_OPT5_SP_WORD4 *)
    R102_1_1_M_차종_SP1 AT %MW10050.0 : BOOL; (* R102_1_1_M_차종_SP1 *)
    R102_1_1_M_차종_SP2 AT %MW10050.1 : BOOL; (* R102_1_1_M_차종_SP2 *)
    R102_1_1_M_차종_SP3 AT %MW10050.2 : BOOL; (* R102_1_1_M_차종_SP3 *)
    R102_1_1_M_차종_SP4 AT %MW10050.3 : BOOL; (* R102_1_1_M_차종_SP4 *)
    R102_1_1_M_차종_SP5 AT %MW10050.4 : BOOL; (* R102_1_1_M_차종_SP5 *)
    R102_1_1_M_차종_SP6 AT %MW10050.5 : BOOL; (* R102_1_1_M_차종_SP6 *)
    R102_1_1_M_차종_SP7 AT %MW10050.6 : BOOL; (* R102_1_1_M_차종_SP7 *)
    R102_1_1_M_차종_SP8 AT %MW10050.7 : BOOL; (* R102_1_1_M_차종_SP8 *)
    R102_1_1_M_차종_SP9 AT %MW10050.15 : BOOL; (* R102_1_1_M_차종_SP9 *)
    R102_1_1_M_차종_공대차 AT %MW10050.12 : BOOL; (* R102_1_1_M_차종_공대차 *)
    R102_1_1_M_차종_공차 AT %MW10050.10 : BOOL; (* R102_1_1_M_차종_공차 *)
    R102_1_1_M_차종_불량대차 AT %MW10050.13 : BOOL; (* R102_1_1_M_차종_불량대차 *)
    R102_1_1_M_차종_불량차 AT %MW10050.11 : BOOL; (* R102_1_1_M_차종_불량차 *)
    R102_1_1_M_차종_비축 AT %MW10050.8 : BOOL; (* R102_1_1_M_차종_비축 *)
    R102_1_1_M_차종_취출대차 AT %MW10050.14 : BOOL; (* R102_1_1_M_차종_취출대차 *)
    R102_1_1_O_RB_0_5S_통신_CHK AT %MW94093.14 : BOOL;
    R102_1_1_O_RB_2차_진입OK AT %MW94091.8 : BOOL;
    R102_1_1_O_RB_3차_진입OK AT %MW94091.9 : BOOL;
    R102_1_1_O_RB_4차_진입OK AT %MW94091.10 : BOOL;
    R102_1_1_O_RB_5차_진입OK AT %MW94091.11 : BOOL;
    R102_1_1_O_RB_6차_진입OK AT %MW94091.12 : BOOL;
    R102_1_1_O_RB_7차_진입OK AT %MW94091.13 : BOOL;
    R102_1_1_O_RB_AX_1차_진입OK AT %MW94091.0 : BOOL;
    R102_1_1_O_RB_B_1차_진입OK AT %MW94091.1 : BOOL;
    R102_1_1_O_RB_C_1차_진입OK AT %MW94091.2 : BOOL;
    R102_1_1_O_RB_D_1차_진입OK AT %MW94091.3 : BOOL;
    R102_1_1_O_RB_EACH_작업완료_리셋 AT %MW94090.14 : BOOL;
    R102_1_1_O_RB_EXT_READY AT %MW94090.11 : BOOL;
    R102_1_1_O_RB_E_1차_진입OK AT %MW94091.4 : BOOL;
    R102_1_1_O_RB_F_1차_진입OK AT %MW94091.5 : BOOL;
    R102_1_1_O_RB_GATE_OPEN_NC AT %MW94093.11 : BOOL;
    R102_1_1_O_RB_G_1차_진입OK AT %MW94091.6 : BOOL;
    R102_1_1_O_RB_H_1차_진입OK AT %MW94091.7 : BOOL;
    R102_1_1_O_RB_MUTUAL_INT1 AT %MW94093.0 : BOOL;
    R102_1_1_O_RB_MUTUAL_INT2 AT %MW94093.1 : BOOL;
    R102_1_1_O_RB_MUTUAL_INT3 AT %MW94093.2 : BOOL;
    R102_1_1_O_RB_MUTUAL_INT4 AT %MW94093.3 : BOOL;
    R102_1_1_O_RB_MUTUAL_INT5 AT %MW94093.4 : BOOL;
    R102_1_1_O_RB_MUTUAL_INT6 AT %MW94093.5 : BOOL;
    R102_1_1_O_RB_MUTUAL_INT7 AT %MW94093.6 : BOOL;
    R102_1_1_O_RB_MUTUAL_INT8 AT %MW94093.7 : BOOL;
    R102_1_1_O_RB_OUTPUT AT %MW94090 : ARRAY[0..3] OF WORD;
    R102_1_1_O_RB_PAUSE_NC AT %MW94090.13 : BOOL;
    R102_1_1_O_RB_PLT10_진입OK AT %MW94092.9 : BOOL;
    R102_1_1_O_RB_PLT11_진입OK AT %MW94092.10 : BOOL;
    R102_1_1_O_RB_PLT12_진입OK AT %MW94092.11 : BOOL;
    R102_1_1_O_RB_PLT1_진입OK AT %MW94092.0 : BOOL;
    R102_1_1_O_RB_PLT2_진입OK AT %MW94092.1 : BOOL;
    R102_1_1_O_RB_PLT3_진입OK AT %MW94092.2 : BOOL;
    R102_1_1_O_RB_PLT4_진입OK AT %MW94092.3 : BOOL;
    R102_1_1_O_RB_PLT5_진입OK AT %MW94092.4 : BOOL;
    R102_1_1_O_RB_PLT6_진입OK AT %MW94092.5 : BOOL;
    R102_1_1_O_RB_PLT7_진입OK AT %MW94092.6 : BOOL;
    R102_1_1_O_RB_PLT8_진입OK AT %MW94092.7 : BOOL;
    R102_1_1_O_RB_PLT9_진입OK AT %MW94092.8 : BOOL;
    R102_1_1_O_RB_PLT_COUNT_리셋_COND AT %MW94093.10 : BOOL;
    R102_1_1_O_RB_PROG_선택1 AT %MW94090.0 : BOOL;
    R102_1_1_O_RB_PROG_선택128 AT %MW94090.7 : BOOL;
    R102_1_1_O_RB_PROG_선택16 AT %MW94090.4 : BOOL;
    R102_1_1_O_RB_PROG_선택2 AT %MW94090.1 : BOOL;
    R102_1_1_O_RB_PROG_선택32 AT %MW94090.5 : BOOL;
    R102_1_1_O_RB_PROG_선택4 AT %MW94090.2 : BOOL;
    R102_1_1_O_RB_PROG_선택64 AT %MW94090.6 : BOOL;
    R102_1_1_O_RB_PROG_선택8 AT %MW94090.3 : BOOL;
    R102_1_1_O_RB_SP_1_14 AT %MW94091.14 : BOOL;
    R102_1_1_O_RB_SP_1_15 AT %MW94091.15 : BOOL;
    R102_1_1_O_RB_SP_2_12 AT %MW94092.12 : BOOL;
    R102_1_1_O_RB_SP_2_13 AT %MW94092.13 : BOOL;
    R102_1_1_O_RB_SP_2_14 AT %MW94092.14 : BOOL;
    R102_1_1_O_RB_SP_5000TH_ON AT %MW94092.15 : BOOL;
    R102_1_1_O_RB_TIP_CHANGE_END AT %MW94093.9 : BOOL;
    R102_1_1_O_RB_TIP_CHANGE_START AT %MW94093.8 : BOOL;
    R102_1_1_O_RB_TIP_DRESS_SATRT AT %MW94090.12 : BOOL;
    R102_1_1_O_RB_VIP_MODE AT %MW94093.15 : BOOL;
    R102_1_1_O_RB_기동 AT %MW94090.9 : BOOL;
    R102_1_1_O_RB_냉각수차단 AT %MW94090.15 : BOOL;
    R102_1_1_O_RB_부저정지 AT %MW94093.13 : BOOL;
    R102_1_1_O_RB_비상정지_NC AT %MW94093.12 : BOOL;
    R102_1_1_O_RB_이상_리셋 AT %MW94090.10 : BOOL;
    R102_1_1_O_RB_작업완료_리셋 AT %MW94090.8 : BOOL;
    R102_1_1_S102_CTYPE_MOVE : FB407_Car_Type_Move_Stn_v1;
    R102_1_1_S103_CTYPE_MOVE : FB407_Car_Type_Move_Stn_v1;
    R102_1_CTYPE_CLEAR : FB409_Car_Type_Clear_v1;
    R102_1_I_RB_0_5_COMM_CHK AT %MW84083.14 : BOOL;
    R102_1_I_RB_10차_간섭무 AT %MW84081.9 : BOOL;
    R102_1_I_RB_11차_간섭무 AT %MW84081.10 : BOOL;
    R102_1_I_RB_12차_간섭무 AT %MW84081.11 : BOOL;
    R102_1_I_RB_1차_간섭무 AT %MW84081.0 : BOOL;
    R102_1_I_RB_1차_작업완료 AT %MW84080.9 : BOOL;
    R102_1_I_RB_2차_간섭무 AT %MW84081.1 : BOOL;
    R102_1_I_RB_2차_작업완료 AT %MW84080.10 : BOOL;
    R102_1_I_RB_3차_간섭무 AT %MW84081.2 : BOOL;
    R102_1_I_RB_3차_작업완료 AT %MW84080.11 : BOOL;
    R102_1_I_RB_4차_간섭무 AT %MW84081.3 : BOOL;
    R102_1_I_RB_4차_작업완료 AT %MW84080.12 : BOOL;
    R102_1_I_RB_5차_간섭무 AT %MW84081.4 : BOOL;
    R102_1_I_RB_5차_작업완료 AT %MW84080.13 : BOOL;
    R102_1_I_RB_6차_간섭무 AT %MW84081.5 : BOOL;
    R102_1_I_RB_6차_작업완료 AT %MW84080.14 : BOOL;
    R102_1_I_RB_7차_간섭무 AT %MW84081.6 : BOOL;
    R102_1_I_RB_7차_작업완료 AT %MW84080.15 : BOOL;
    R102_1_I_RB_8차_간섭무 AT %MW84081.7 : BOOL;
    R102_1_I_RB_9차_간섭무 AT %MW84081.8 : BOOL;
    R102_1_I_RB_AB_NORMAL_선택 AT %MW84080.6 : BOOL;
    R102_1_I_RB_GUN1_FIXED_TIP AT %MW84087 : WORD;
    R102_1_I_RB_GUN1_MOVING_TIP AT %MW84086 : WORD;
    R102_1_I_RB_GUN2_FIXED_TIP AT %MW84089 : WORD;
    R102_1_I_RB_GUN2_MOVING_TIP AT %MW84088 : WORD;
    R102_1_I_RB_INPUT AT %MW84080 : ARRAY[0..3] OF WORD;
    R102_1_I_RB_LS_이상 AT %MW84082.11 : BOOL;
    R102_1_I_RB_MOTOR_MC_ON AT %MW84083.15 : BOOL;
    R102_1_I_RB_MUTUAL_INT1 AT %MW84083.0 : BOOL;
    R102_1_I_RB_MUTUAL_INT2 AT %MW84083.1 : BOOL;
    R102_1_I_RB_MUTUAL_INT3 AT %MW84083.2 : BOOL;
    R102_1_I_RB_MUTUAL_INT4 AT %MW84083.3 : BOOL;
    R102_1_I_RB_MUTUAL_INT5 AT %MW84083.4 : BOOL;
    R102_1_I_RB_MUTUAL_INT6 AT %MW84083.5 : BOOL;
    R102_1_I_RB_MUTUAL_INT7 AT %MW84083.6 : BOOL;
    R102_1_I_RB_MUTUAL_INT8 AT %MW84083.7 : BOOL;
    R102_1_I_RB_PLT_UNLOAD_완료 AT %MW84083.11 : BOOL;
    R102_1_I_RB_PLT_최종UNLOAD_완료 AT %MW84083.12 : BOOL;
    R102_1_I_RB_PROG_ECHO_1 AT %MW84082.0 : BOOL;
    R102_1_I_RB_PROG_ECHO_128 AT %MW84082.7 : BOOL;
    R102_1_I_RB_PROG_ECHO_16 AT %MW84082.4 : BOOL;
    R102_1_I_RB_PROG_ECHO_2 AT %MW84082.1 : BOOL;
    R102_1_I_RB_PROG_ECHO_32 AT %MW84082.5 : BOOL;
    R102_1_I_RB_PROG_ECHO_4 AT %MW84082.2 : BOOL;
    R102_1_I_RB_PROG_ECHO_64 AT %MW84082.6 : BOOL;
    R102_1_I_RB_PROG_ECHO_8 AT %MW84082.3 : BOOL;
    R102_1_I_RB_SP3_8 AT %MW84083.8 : BOOL;
    R102_1_I_RB_SP3_9 AT %MW84083.9 : BOOL;
    R102_1_I_RB_SPARE_WORD_4 AT %MW84084 : WORD;
    R102_1_I_RB_SP_1_12 AT %MW84081.12 : BOOL;
    R102_1_I_RB_SP_1_13 AT %MW84081.13 : BOOL;
    R102_1_I_RB_SP_1_14 AT %MW84081.14 : BOOL;
    R102_1_I_RB_SP_1_15 AT %MW84081.15 : BOOL;
    R102_1_I_RB_TC_이상 AT %MW84082.8 : BOOL;
    R102_1_I_RB_TIP_CHANGE AT %MW84083.13 : BOOL;
    R102_1_I_RB_TIP_DRESSING AT %MW84080.7 : BOOL;
    R102_1_I_RB__PLT_카운터리셋완료 AT %MW84083.10 : BOOL;
    R102_1_I_RB_공기압_이상 AT %MW84082.9 : BOOL;
    R102_1_I_RB_냉각수_이상 AT %MW84082.10 : BOOL;
    R102_1_I_RB_비상정지_NC AT %MW84080.8 : BOOL;
    R102_1_I_RB_비전이상 AT %MW84082.14 : BOOL;
    R102_1_I_RB_실러이상 AT %MW84082.13 : BOOL;
    R102_1_I_RB_용접카운터이상 AT %MW84082.15 : BOOL;
    R102_1_I_RB_용접타점수 AT %MW84085 : WORD;
    R102_1_I_RB_운전준비 AT %MW84080.3 : BOOL;
    R102_1_I_RB_원위치 AT %MW84080.0 : BOOL;
    R102_1_I_RB_이상리셋 AT %MW84080.2 : BOOL;
    R102_1_I_RB_자동 AT %MW84080.4 : BOOL;
    R102_1_I_RB_자동기동 AT %MW84080.5 : BOOL;
    R102_1_I_RB_최종_작업완료 AT %MW84080.1 : BOOL;
    R102_1_I_RB_통신이상 AT %MW84082.12 : BOOL;
    R102_1_M_DATA_삭제_PLS AT %MW9004.0 : BOOL; (* R102_1_M_DATA_삭제_PLS *)
    R102_1_M_DATA_삭제_SIGN AT %MW9004.1 : BOOL; (* R102_1_M_DATA_삭제_SIGN *)
    R102_1_M_DATA_삭제_완료 AT %MW9004.2 : BOOL; (* R102_1_M_DATA_삭제_완료 *)
    R102_1_M_DATA_전송_MEMO AT %MW9004.8 : BOOL; (* R102_1_M_DATA_전송_MEMO *)
    R102_1_M_DATA_전송_PLS AT %MW9004.9 : BOOL; (* R102_1_M_DATA_전송_PLS *)
    R102_1_M_DATA_전송_SIGN AT %MW9004.10 : BOOL; (* R102_1_M_DATA_전송_SIGN *)
    R102_1_M_DATA_전송_완료 AT %MW9004.11 : BOOL; (* R102_1_M_DATA_전송_완료 *)
    R102_1_M_I_RB_1차_작업완료 AT %MW20081.2 : BOOL;
    R102_1_M_I_RB_2차_작업완료 AT %MW20081.3 : BOOL;
    R102_1_M_I_RB_3차_작업완료 AT %MW20081.4 : BOOL;
    R102_1_M_I_RB_4차_작업완료 AT %MW20081.5 : BOOL;
    R102_1_M_I_RB_5차_작업완료 AT %MW20081.6 : BOOL;
    R102_1_M_I_RB_6차_작업완료 AT %MW20081.7 : BOOL;
    R102_1_M_I_RB_7차_작업완료 AT %MW20081.8 : BOOL;
    R102_1_M_I_RB_PAUSE_보조 AT %MW20080.5 : BOOL;
    R102_1_M_I_RB_PLC_RUN_CHK_이상 AT %MW20080.7 : BOOL;
    R102_1_M_I_RB_간섭무_1 AT %MW20082.0 : BOOL;
    R102_1_M_I_RB_간섭무_10 AT %MW20082.9 : BOOL;
    R102_1_M_I_RB_간섭무_11 AT %MW20082.10 : BOOL;
    R102_1_M_I_RB_간섭무_12 AT %MW20082.11 : BOOL;
    R102_1_M_I_RB_간섭무_2 AT %MW20082.1 : BOOL;
    R102_1_M_I_RB_간섭무_3 AT %MW20082.2 : BOOL;
    R102_1_M_I_RB_간섭무_4 AT %MW20082.3 : BOOL;
    R102_1_M_I_RB_간섭무_5 AT %MW20082.4 : BOOL;
    R102_1_M_I_RB_간섭무_6 AT %MW20082.5 : BOOL;
    R102_1_M_I_RB_간섭무_7 AT %MW20082.6 : BOOL;
    R102_1_M_I_RB_간섭무_8 AT %MW20082.7 : BOOL;
    R102_1_M_I_RB_간섭무_9 AT %MW20082.8 : BOOL;
    R102_1_M_I_RB_비상정지 AT %MW20080.4 : BOOL;
    R102_1_M_I_RB_운전준비 AT %MW20080.0 : BOOL;
    R102_1_M_I_RB_원위치 AT %MW20080.3 : BOOL;
    R102_1_M_I_RB_이상 AT %MW20080.2 : BOOL;
    R102_1_M_I_RB_자동 AT %MW20080.1 : BOOL;
    R102_1_M_I_RB_최종작업완료 AT %MW20081.0 : BOOL;
    R102_1_M_I_RB_프로그램_이상 AT %MW20080.6 : BOOL;
    R102_1_M_O_RB_1_CYCLE_SET AT %MW21080.3 : BOOL;
    R102_1_M_O_RB_1_CYCLE_리셋 AT %MW21080.4 : BOOL;
    R102_1_M_O_RB_1차_작업완료_리셋 AT %MW21082.0 : BOOL;
    R102_1_M_O_RB_2차_작업완료_리셋 AT %MW21082.1 : BOOL;
    R102_1_M_O_RB_2차_진입OK AT %MW21081.8 : BOOL;
    R102_1_M_O_RB_3차_작업완료_리셋 AT %MW21082.2 : BOOL;
    R102_1_M_O_RB_3차_진입OK AT %MW21081.9 : BOOL;
    R102_1_M_O_RB_4차_작업완료_리셋 AT %MW21082.3 : BOOL;
    R102_1_M_O_RB_4차_진입OK AT %MW21081.10 : BOOL;
    R102_1_M_O_RB_5차_작업완료_리셋 AT %MW21082.4 : BOOL;
    R102_1_M_O_RB_5차_진입OK AT %MW21081.11 : BOOL;
    R102_1_M_O_RB_6차_작업완료_리셋 AT %MW21082.5 : BOOL;
    R102_1_M_O_RB_6차_진입OK AT %MW21081.12 : BOOL;
    R102_1_M_O_RB_7차_작업완료_리셋 AT %MW21082.6 : BOOL;
    R102_1_M_O_RB_7차_진입OK AT %MW21081.13 : BOOL;
    R102_1_M_O_RB_ATD_OK AT %MW21080.6 : BOOL;
    R102_1_M_O_RB_PLT_10_진입OK AT %MW21083.10 : BOOL;
    R102_1_M_O_RB_PLT_11_진입OK AT %MW21083.11 : BOOL;
    R102_1_M_O_RB_PLT_12_진입OK AT %MW21083.12 : BOOL;
    R102_1_M_O_RB_PLT_1_진입OK AT %MW21083.1 : BOOL;
    R102_1_M_O_RB_PLT_2_진입OK AT %MW21083.2 : BOOL;
    R102_1_M_O_RB_PLT_3_진입OK AT %MW21083.3 : BOOL;
    R102_1_M_O_RB_PLT_4_진입OK AT %MW21083.4 : BOOL;
    R102_1_M_O_RB_PLT_5_진입OK AT %MW21083.5 : BOOL;
    R102_1_M_O_RB_PLT_6_진입OK AT %MW21083.6 : BOOL;
    R102_1_M_O_RB_PLT_7_진입OK AT %MW21083.7 : BOOL;
    R102_1_M_O_RB_PLT_8_진입OK AT %MW21083.8 : BOOL;
    R102_1_M_O_RB_PLT_9_진입OK AT %MW21083.9 : BOOL;
    R102_1_M_O_RB_PLT_카운터리셋_보조 AT %MW21080.10 : BOOL;
    R102_1_M_O_RB_RESTART_OK AT %MW21080.2 : BOOL;
    R102_1_M_O_RB_START_OK AT %MW21080.0 : BOOL;
    R102_1_M_O_RB_TEST_MODE_5000회 AT %MW21080.12 : BOOL;
    R102_1_M_O_RB_TIP_교체_시작 AT %MW21080.7 : BOOL;
    R102_1_M_O_RB_TIP_교체_완료 AT %MW21080.8 : BOOL;
    R102_1_M_O_RB_VIP_MODE AT %MW21080.11 : BOOL;
    R102_1_M_O_RB_냉각수_차단_요청 AT %MW21080.9 : BOOL;
    R102_1_M_O_RB_진입OK_AX차종 AT %MW21081.0 : BOOL;
    R102_1_M_O_RB_진입OK_B차종 AT %MW21081.1 : BOOL;
    R102_1_M_O_RB_진입OK_C차종 AT %MW21081.2 : BOOL;
    R102_1_M_O_RB_진입OK_D차종 AT %MW21081.3 : BOOL;
    R102_1_M_O_RB_진입OK_E차종 AT %MW21081.4 : BOOL;
    R102_1_M_O_RB_진입OK_F차종 AT %MW21081.5 : BOOL;
    R102_1_M_O_RB_진입OK_G차종 AT %MW21081.6 : BOOL;
    R102_1_M_O_RB_진입OK_H차종 AT %MW21081.7 : BOOL;
    R102_1_M_O_RB_최종_작업완료_리셋 AT %MW21080.5 : BOOL;
    R102_1_M_O_RB_프로그램_OK AT %MW21080.1 : BOOL;
    R102_1_M_RB_PROG_NO AT %MW20084 : WORD;
    R102_1_M_RB_통신이상 AT %MW1524.4 : BOOL;
    R102_1_M_SEQ AT %MW10080 : WORD; (* R102_1_M_SEQ *)
    R102_1_M_STN_차종_NONE AT %MW1502.5 : BOOL;
    R102_1_M_STN_차종_ON AT %MW1502.4 : BOOL;
    R102_1_M_VIN_NO_1_2 AT %MW10091 : WORD; (* R102_1_M_VIN_NO_1_2 *)
    R102_1_M_VIN_NO_3_4 AT %MW10092 : WORD; (* R102_1_M_VIN_NO_3_4 *)
    R102_1_M_VIN_NO_5_6 AT %MW10093 : WORD; (* R102_1_M_VIN_NO_5_6 *)
    R102_1_M_VIN_NO_7_8 AT %MW10094 : WORD; (* R102_1_M_VIN_NO_7_8 *)
    R102_1_M_VIN_NO_9_10 AT %MW10095 : WORD; (* R102_1_M_VIN_NO_9_10 *)
    R102_1_M_차종1_AX AT %MW10081.0 : BOOL; (* R102_1_M_차종1_AX *)
    R102_1_M_차종1_B AT %MW10081.1 : BOOL; (* R102_1_M_차종1_B *)
    R102_1_M_차종1_C AT %MW10081.2 : BOOL; (* R102_1_M_차종1_C *)
    R102_1_M_차종1_D AT %MW10081.3 : BOOL; (* R102_1_M_차종1_D *)
    R102_1_M_차종1_E AT %MW10081.4 : BOOL; (* R102_1_M_차종1_E *)
    R102_1_M_차종1_F AT %MW10081.5 : BOOL; (* R102_1_M_차종1_F *)
    R102_1_M_차종1_G AT %MW10081.6 : BOOL; (* R102_1_M_차종1_G *)
    R102_1_M_차종1_H AT %MW10081.7 : BOOL; (* R102_1_M_차종1_H *)
    R102_1_M_차종2_3DR AT %MW10081.8 : BOOL; (* R102_1_M_차종2_3DR *)
    R102_1_M_차종2_4DR AT %MW10081.9 : BOOL; (* R102_1_M_차종2_4DR *)
    R102_1_M_차종2_5DR AT %MW10081.10 : BOOL; (* R102_1_M_차종2_5DR *)
    R102_1_M_차종2_SP1 AT %MW10081.12 : BOOL; (* R102_1_M_차종2_SP1 *)
    R102_1_M_차종2_SP2 AT %MW10081.13 : BOOL; (* R102_1_M_차종2_SP2 *)
    R102_1_M_차종2_WGN AT %MW10081.11 : BOOL; (* R102_1_M_차종2_WGN *)
    R102_1_M_차종3_LHD AT %MW10081.14 : BOOL; (* R102_1_M_차종3_LHD *)
    R102_1_M_차종3_RHD AT %MW10081.15 : BOOL; (* R102_1_M_차종3_RHD *)
    R102_1_M_차종4_EEC AT %MW10082.3 : BOOL; (* R102_1_M_차종4_EEC *)
    R102_1_M_차종4_SP1 AT %MW10082.8 : BOOL; (* R102_1_M_차종4_SP1 *)
    R102_1_M_차종4_SP2 AT %MW10082.9 : BOOL; (* R102_1_M_차종4_SP2 *)
    R102_1_M_차종4_SP3 AT %MW10082.11 : BOOL; (* R102_1_M_차종4_SP3 *)
    R102_1_M_차종4_SP4 AT %MW10082.12 : BOOL; (* R102_1_M_차종4_SP4 *)
    R102_1_M_차종4_SP5 AT %MW10082.13 : BOOL; (* R102_1_M_차종4_SP5 *)
    R102_1_M_차종4_SP6 AT %MW10082.14 : BOOL; (* R102_1_M_차종4_SP6 *)
    R102_1_M_차종4_SP7 AT %MW10082.15 : BOOL; (* R102_1_M_차종4_SP7 *)
    R102_1_M_차종4_내수 AT %MW10082.0 : BOOL; (* R102_1_M_차종4_내수 *)
    R102_1_M_차종4_러시아 AT %MW10082.10 : BOOL; (* R102_1_M_차종4_러시아 *)
    R102_1_M_차종4_북미 AT %MW10082.2 : BOOL; (* R102_1_M_차종4_북미 *)
    R102_1_M_차종4_브라질 AT %MW10082.7 : BOOL; (* R102_1_M_차종4_브라질 *)
    R102_1_M_차종4_수출 AT %MW10082.1 : BOOL; (* R102_1_M_차종4_수출 *)
    R102_1_M_차종4_중국 AT %MW10082.6 : BOOL; (* R102_1_M_차종4_중국 *)
    R102_1_M_차종4_중동 AT %MW10082.5 : BOOL; (* R102_1_M_차종4_중동 *)
    R102_1_M_차종4_호주 AT %MW10082.4 : BOOL; (* R102_1_M_차종4_호주 *)
    R102_1_M_차종5_AT AT %MW10083.1 : BOOL; (* R102_1_M_차종5_AT *)
    R102_1_M_차종5_MT AT %MW10083.0 : BOOL; (* R102_1_M_차종5_MT *)
    R102_1_M_차종5_SP1 AT %MW10083.2 : BOOL; (* R102_1_M_차종5_SP1 *)
    R102_1_M_차종6_DSROOF AT %MW10083.6 : BOOL; (* R102_1_M_차종6_DSROOF *)
    R102_1_M_차종6_SP1 AT %MW10083.7 : BOOL; (* R102_1_M_차종6_SP1 *)
    R102_1_M_차종6_썬루프 AT %MW10083.4 : BOOL; (* R102_1_M_차종6_썬루프 *)
    R102_1_M_차종6_일반루프 AT %MW10083.3 : BOOL; (* R102_1_M_차종6_일반루프 *)
    R102_1_M_차종6_파노라마루프 AT %MW10083.5 : BOOL; (* R102_1_M_차종6_파노라마루프 *)
    R102_1_M_차종7_DSL AT %MW10083.9 : BOOL; (* R102_1_M_차종7_DSL *)
    R102_1_M_차종7_GSL AT %MW10083.8 : BOOL; (* R102_1_M_차종7_GSL *)
    R102_1_M_차종7_SP1 AT %MW10083.10 : BOOL; (* R102_1_M_차종7_SP1 *)
    R102_1_M_차종7_SP2 AT %MW10083.11 : BOOL; (* R102_1_M_차종7_SP2 *)
    R102_1_M_차종7_SP3 AT %MW10083.12 : BOOL; (* R102_1_M_차종7_SP3 *)
    R102_1_M_차종7_SP4 AT %MW10083.13 : BOOL; (* R102_1_M_차종7_SP4 *)
    R102_1_M_차종7_SP5 AT %MW10083.14 : BOOL; (* R102_1_M_차종7_SP5 *)
    R102_1_M_차종7_SP6 AT %MW10083.15 : BOOL; (* R102_1_M_차종7_SP6 *)
    R102_1_M_차종8_2WD AT %MW10084.0 : BOOL; (* R102_1_M_차종8_2WD *)
    R102_1_M_차종8_4WD AT %MW10084.1 : BOOL; (* R102_1_M_차종8_4WD *)
    R102_1_M_차종8_SP1 AT %MW10084.2 : BOOL; (* R102_1_M_차종8_SP1 *)
    R102_1_M_차종9_MPI AT %MW10084.3 : BOOL; (* R102_1_M_차종9_MPI *)
    R102_1_M_차종9_SP1 AT %MW10084.5 : BOOL; (* R102_1_M_차종9_SP1 *)
    R102_1_M_차종9_SP10 AT %MW10084.14 : BOOL; (* R102_1_M_차종9_SP10 *)
    R102_1_M_차종9_SP11 AT %MW10084.15 : BOOL; (* R102_1_M_차종9_SP11 *)
    R102_1_M_차종9_SP2 AT %MW10084.6 : BOOL; (* R102_1_M_차종9_SP2 *)
    R102_1_M_차종9_SP3 AT %MW10084.7 : BOOL; (* R102_1_M_차종9_SP3 *)
    R102_1_M_차종9_SP4 AT %MW10084.8 : BOOL; (* R102_1_M_차종9_SP4 *)
    R102_1_M_차종9_SP5 AT %MW10084.9 : BOOL; (* R102_1_M_차종9_SP5 *)
    R102_1_M_차종9_SP6 AT %MW10084.10 : BOOL; (* R102_1_M_차종9_SP6 *)
    R102_1_M_차종9_SP7 AT %MW10084.11 : BOOL; (* R102_1_M_차종9_SP7 *)
    R102_1_M_차종9_SP8 AT %MW10084.12 : BOOL; (* R102_1_M_차종9_SP8 *)
    R102_1_M_차종9_SP9 AT %MW10084.13 : BOOL; (* R102_1_M_차종9_SP9 *)
    R102_1_M_차종9_T_GDI AT %MW10084.4 : BOOL; (* R102_1_M_차종9_T_GDI *)
    R102_1_M_차종_AS AT %MW10090.9 : BOOL; (* R102_1_M_차종_AS *)
    R102_1_M_차종_MATCH_이상 AT %MW1015.1 : BOOL;
    R102_1_M_차종_OPT1_R_RACK_무 AT %MW10085.3 : BOOL; (* R102_1_M_차종_OPT1_R_RACK_무 *)
    R102_1_M_차종_OPT1_R_RACK_유 AT %MW10085.2 : BOOL; (* R102_1_M_차종_OPT1_R_RACK_유 *)
    R102_1_M_차종_OPT1_SP1 AT %MW10085.10 : BOOL; (* R102_1_M_차종_OPT1_SP1 *)
    R102_1_M_차종_OPT1_SP2 AT %MW10085.11 : BOOL; (* R102_1_M_차종_OPT1_SP2 *)
    R102_1_M_차종_OPT1_SP3 AT %MW10085.12 : BOOL; (* R102_1_M_차종_OPT1_SP3 *)
    R102_1_M_차종_OPT1_SP4 AT %MW10085.13 : BOOL; (* R102_1_M_차종_OPT1_SP4 *)
    R102_1_M_차종_OPT1_SP5 AT %MW10085.14 : BOOL; (* R102_1_M_차종_OPT1_SP5 *)
    R102_1_M_차종_OPT1_SP6 AT %MW10085.15 : BOOL; (* R102_1_M_차종_OPT1_SP6 *)
    R102_1_M_차종_OPT1_S_REP_EATER_무 AT %MW10085.7 : BOOL; (* R102_1_M_차종_OPT1_S_REP_EATER_무 *)
    R102_1_M_차종_OPT1_S_REP_EATER_유 AT %MW10085.6 : BOOL; (* R102_1_M_차종_OPT1_S_REP_EATER_유 *)
    R102_1_M_차종_OPT1_VAN_무 AT %MW10085.9 : BOOL; (* R102_1_M_차종_OPT1_VAN_무 *)
    R102_1_M_차종_OPT1_VAN_유 AT %MW10085.8 : BOOL; (* R102_1_M_차종_OPT1_VAN_유 *)
    R102_1_M_차종_OPT1_슬라이딩_무 AT %MW10085.1 : BOOL; (* R102_1_M_차종_OPT1_슬라이딩_무 *)
    R102_1_M_차종_OPT1_슬라이딩_유 AT %MW10085.0 : BOOL; (* R102_1_M_차종_OPT1_슬라이딩_유 *)
    R102_1_M_차종_OPT1_폴딩_무 AT %MW10085.5 : BOOL; (* R102_1_M_차종_OPT1_폴딩_무 *)
    R102_1_M_차종_OPT1_폴딩_유 AT %MW10085.4 : BOOL; (* R102_1_M_차종_OPT1_폴딩_유 *)
    R102_1_M_차종_OPT2_SP_WORD1 AT %MW10086 : WORD; (* R102_1_M_차종_OPT2_SP_WORD1 *)
    R102_1_M_차종_OPT3_SP_WORD2 AT %MW10087 : WORD; (* R102_1_M_차종_OPT3_SP_WORD2 *)
    R102_1_M_차종_OPT4_SP_WORD3 AT %MW10088 : WORD; (* R102_1_M_차종_OPT4_SP_WORD3 *)
    R102_1_M_차종_OPT5_SP_WORD4 AT %MW10089 : WORD; (* R102_1_M_차종_OPT5_SP_WORD4 *)
    R102_1_M_차종_SP1 AT %MW10090.0 : BOOL; (* R102_1_M_차종_SP1 *)
    R102_1_M_차종_SP2 AT %MW10090.1 : BOOL; (* R102_1_M_차종_SP2 *)
    R102_1_M_차종_SP3 AT %MW10090.2 : BOOL; (* R102_1_M_차종_SP3 *)
    R102_1_M_차종_SP4 AT %MW10090.3 : BOOL; (* R102_1_M_차종_SP4 *)
    R102_1_M_차종_SP5 AT %MW10090.4 : BOOL; (* R102_1_M_차종_SP5 *)
    R102_1_M_차종_SP6 AT %MW10090.5 : BOOL; (* R102_1_M_차종_SP6 *)
    R102_1_M_차종_SP7 AT %MW10090.6 : BOOL; (* R102_1_M_차종_SP7 *)
    R102_1_M_차종_SP8 AT %MW10090.7 : BOOL; (* R102_1_M_차종_SP8 *)
    R102_1_M_차종_SP9 AT %MW10090.15 : BOOL; (* R102_1_M_차종_SP9 *)
    R102_1_M_차종_공대차 AT %MW10090.12 : BOOL; (* R102_1_M_차종_공대차 *)
    R102_1_M_차종_공차 AT %MW10090.10 : BOOL; (* R102_1_M_차종_공차 *)
    R102_1_M_차종_불량대차 AT %MW10090.13 : BOOL; (* R102_1_M_차종_불량대차 *)
    R102_1_M_차종_불량차 AT %MW10090.11 : BOOL; (* R102_1_M_차종_불량차 *)
    R102_1_M_차종_비축 AT %MW10090.8 : BOOL; (* R102_1_M_차종_비축 *)
    R102_1_M_차종_취출대차 AT %MW10090.14 : BOOL; (* R102_1_M_차종_취출대차 *)
    R102_1_O_RB_0_5S_통신_CHK AT %MW94083.14 : BOOL;
    R102_1_O_RB_2차_진입OK AT %MW94081.8 : BOOL;
    R102_1_O_RB_3차_진입OK AT %MW94081.9 : BOOL;
    R102_1_O_RB_4차_진입OK AT %MW94081.10 : BOOL;
    R102_1_O_RB_5차_진입OK AT %MW94081.11 : BOOL;
    R102_1_O_RB_6차_진입OK AT %MW94081.12 : BOOL;
    R102_1_O_RB_7차_진입OK AT %MW94081.13 : BOOL;
    R102_1_O_RB_AX_1차_진입OK AT %MW94081.0 : BOOL;
    R102_1_O_RB_B_1차_진입OK AT %MW94081.1 : BOOL;
    R102_1_O_RB_C_1차_진입OK AT %MW94081.2 : BOOL;
    R102_1_O_RB_D_1차_진입OK AT %MW94081.3 : BOOL;
    R102_1_O_RB_EACH_작업완료_리셋 AT %MW94080.14 : BOOL;
    R102_1_O_RB_EXT_READY AT %MW94080.11 : BOOL;
    R102_1_O_RB_E_1차_진입OK AT %MW94081.4 : BOOL;
    R102_1_O_RB_F_1차_진입OK AT %MW94081.5 : BOOL;
    R102_1_O_RB_GATE_OPEN_NC AT %MW94083.11 : BOOL;
    R102_1_O_RB_G_1차_진입OK AT %MW94081.6 : BOOL;
    R102_1_O_RB_H_1차_진입OK AT %MW94081.7 : BOOL;
    R102_1_O_RB_MUTUAL_INT1 AT %MW94083.0 : BOOL;
    R102_1_O_RB_MUTUAL_INT2 AT %MW94083.1 : BOOL;
    R102_1_O_RB_MUTUAL_INT3 AT %MW94083.2 : BOOL;
    R102_1_O_RB_MUTUAL_INT4 AT %MW94083.3 : BOOL;
    R102_1_O_RB_MUTUAL_INT5 AT %MW94083.4 : BOOL;
    R102_1_O_RB_MUTUAL_INT6 AT %MW94083.5 : BOOL;
    R102_1_O_RB_MUTUAL_INT7 AT %MW94083.6 : BOOL;
    R102_1_O_RB_MUTUAL_INT8 AT %MW94083.7 : BOOL;
    R102_1_O_RB_OUTPUT AT %MW94080 : ARRAY[0..3] OF WORD;
    R102_1_O_RB_PAUSE_NC AT %MW94080.13 : BOOL;
    R102_1_O_RB_PLT10_진입OK AT %MW94082.9 : BOOL;
    R102_1_O_RB_PLT11_진입OK AT %MW94082.10 : BOOL;
    R102_1_O_RB_PLT12_진입OK AT %MW94082.11 : BOOL;
    R102_1_O_RB_PLT1_진입OK AT %MW94082.0 : BOOL;
    R102_1_O_RB_PLT2_진입OK AT %MW94082.1 : BOOL;
    R102_1_O_RB_PLT3_진입OK AT %MW94082.2 : BOOL;
    R102_1_O_RB_PLT4_진입OK AT %MW94082.3 : BOOL;
    R102_1_O_RB_PLT5_진입OK AT %MW94082.4 : BOOL;
    R102_1_O_RB_PLT6_진입OK AT %MW94082.5 : BOOL;
    R102_1_O_RB_PLT7_진입OK AT %MW94082.6 : BOOL;
    R102_1_O_RB_PLT8_진입OK AT %MW94082.7 : BOOL;
    R102_1_O_RB_PLT9_진입OK AT %MW94082.8 : BOOL;
    R102_1_O_RB_PLT_COUNT_리셋_COND AT %MW94083.10 : BOOL;
    R102_1_O_RB_PROG_선택1 AT %MW94080.0 : BOOL;
    R102_1_O_RB_PROG_선택128 AT %MW94080.7 : BOOL;
    R102_1_O_RB_PROG_선택16 AT %MW94080.4 : BOOL;
    R102_1_O_RB_PROG_선택2 AT %MW94080.1 : BOOL;
    R102_1_O_RB_PROG_선택32 AT %MW94080.5 : BOOL;
    R102_1_O_RB_PROG_선택4 AT %MW94080.2 : BOOL;
    R102_1_O_RB_PROG_선택64 AT %MW94080.6 : BOOL;
    R102_1_O_RB_PROG_선택8 AT %MW94080.3 : BOOL;
    R102_1_O_RB_SP_1_14 AT %MW94081.14 : BOOL;
    R102_1_O_RB_SP_1_15 AT %MW94081.15 : BOOL;
    R102_1_O_RB_SP_2_12 AT %MW94082.12 : BOOL;
    R102_1_O_RB_SP_2_13 AT %MW94082.13 : BOOL;
    R102_1_O_RB_SP_2_14 AT %MW94082.14 : BOOL;
    R102_1_O_RB_SP_5000TH_ON AT %MW94082.15 : BOOL;
    R102_1_O_RB_TIP_CHANGE_END AT %MW94083.9 : BOOL;
    R102_1_O_RB_TIP_CHANGE_START AT %MW94083.8 : BOOL;
    R102_1_O_RB_TIP_DRESS_SATRT AT %MW94080.12 : BOOL;
    R102_1_O_RB_VIP_MODE AT %MW94083.15 : BOOL;
    R102_1_O_RB_기동 AT %MW94080.9 : BOOL;
    R102_1_O_RB_냉각수차단 AT %MW94080.15 : BOOL;
    R102_1_O_RB_부저정지 AT %MW94083.13 : BOOL;
    R102_1_O_RB_비상정지_NC AT %MW94083.12 : BOOL;
    R102_1_O_RB_이상_리셋 AT %MW94080.10 : BOOL;
    R102_1_O_RB_작업완료_리셋 AT %MW94080.8 : BOOL;
    R102_1_S103_CTYPE_MOVE : FB407_Car_Type_Move_Stn_v1;
    R102_1_S104_CTYPE_MOVE : FB407_Car_Type_Move_Stn_v1;
    R102_2_CTYPE_CLEAR : FB409_Car_Type_Clear_v1;
    R103_1_I_RB_0_5_COMM_CHK AT %MW84103.14 : BOOL;
    R103_1_I_RB_10차_간섭무 AT %MW84101.9 : BOOL;
    R103_1_I_RB_11차_간섭무 AT %MW84101.10 : BOOL;
    R103_1_I_RB_12차_간섭무 AT %MW84101.11 : BOOL;
    R103_1_I_RB_1차_간섭무 AT %MW84101.0 : BOOL;
    R103_1_I_RB_1차_작업완료 AT %MW84100.9 : BOOL;
    R103_1_I_RB_2차_간섭무 AT %MW84101.1 : BOOL;
    R103_1_I_RB_2차_작업완료 AT %MW84100.10 : BOOL;
    R103_1_I_RB_3차_간섭무 AT %MW84101.2 : BOOL;
    R103_1_I_RB_3차_작업완료 AT %MW84100.11 : BOOL;
    R103_1_I_RB_4차_간섭무 AT %MW84101.3 : BOOL;
    R103_1_I_RB_4차_작업완료 AT %MW84100.12 : BOOL;
    R103_1_I_RB_5차_간섭무 AT %MW84101.4 : BOOL;
    R103_1_I_RB_5차_작업완료 AT %MW84100.13 : BOOL;
    R103_1_I_RB_6차_간섭무 AT %MW84101.5 : BOOL;
    R103_1_I_RB_6차_작업완료 AT %MW84100.14 : BOOL;
    R103_1_I_RB_7차_간섭무 AT %MW84101.6 : BOOL;
    R103_1_I_RB_7차_작업완료 AT %MW84100.15 : BOOL;
    R103_1_I_RB_8차_간섭무 AT %MW84101.7 : BOOL;
    R103_1_I_RB_9차_간섭무 AT %MW84101.8 : BOOL;
    R103_1_I_RB_AB_NORMAL_선택 AT %MW84100.6 : BOOL;
    R103_1_I_RB_GUN1_FIXED_TIP AT %MW84107 : WORD;
    R103_1_I_RB_GUN1_MOVING_TIP AT %MW84106 : WORD;
    R103_1_I_RB_GUN2_FIXED_TIP AT %MW84109 : WORD;
    R103_1_I_RB_GUN2_MOVING_TIP AT %MW84108 : WORD;
    R103_1_I_RB_INPUT AT %MW84100 : ARRAY[0..3] OF WORD;
    R103_1_I_RB_LS_이상 AT %MW84102.11 : BOOL;
    R103_1_I_RB_MOTOR_MC_ON AT %MW84103.15 : BOOL;
    R103_1_I_RB_MUTUAL_INT1 AT %MW84103.0 : BOOL;
    R103_1_I_RB_MUTUAL_INT2 AT %MW84103.1 : BOOL;
    R103_1_I_RB_MUTUAL_INT3 AT %MW84103.2 : BOOL;
    R103_1_I_RB_MUTUAL_INT4 AT %MW84103.3 : BOOL;
    R103_1_I_RB_MUTUAL_INT5 AT %MW84103.4 : BOOL;
    R103_1_I_RB_MUTUAL_INT6 AT %MW84103.5 : BOOL;
    R103_1_I_RB_MUTUAL_INT7 AT %MW84103.6 : BOOL;
    R103_1_I_RB_MUTUAL_INT8 AT %MW84103.7 : BOOL;
    R103_1_I_RB_PLT_UNLOAD_완료 AT %MW84103.11 : BOOL;
    R103_1_I_RB_PLT_최종UNLOAD_완료 AT %MW84103.12 : BOOL;
    R103_1_I_RB_PROG_ECHO_1 AT %MW84102.0 : BOOL;
    R103_1_I_RB_PROG_ECHO_128 AT %MW84102.7 : BOOL;
    R103_1_I_RB_PROG_ECHO_16 AT %MW84102.4 : BOOL;
    R103_1_I_RB_PROG_ECHO_2 AT %MW84102.1 : BOOL;
    R103_1_I_RB_PROG_ECHO_32 AT %MW84102.5 : BOOL;
    R103_1_I_RB_PROG_ECHO_4 AT %MW84102.2 : BOOL;
    R103_1_I_RB_PROG_ECHO_64 AT %MW84102.6 : BOOL;
    R103_1_I_RB_PROG_ECHO_8 AT %MW84102.3 : BOOL;
    R103_1_I_RB_SP3_8 AT %MW84103.8 : BOOL;
    R103_1_I_RB_SP3_9 AT %MW84103.9 : BOOL;
    R103_1_I_RB_SPARE_WORD_4 AT %MW84104 : WORD;
    R103_1_I_RB_SP_1_12 AT %MW84101.12 : BOOL;
    R103_1_I_RB_SP_1_13 AT %MW84101.13 : BOOL;
    R103_1_I_RB_SP_1_14 AT %MW84101.14 : BOOL;
    R103_1_I_RB_SP_1_15 AT %MW84101.15 : BOOL;
    R103_1_I_RB_TC_이상 AT %MW84102.8 : BOOL;
    R103_1_I_RB_TIP_CHANGE AT %MW84103.13 : BOOL;
    R103_1_I_RB_TIP_DRESSING AT %MW84100.7 : BOOL;
    R103_1_I_RB__PLT_카운터리셋완료 AT %MW84103.10 : BOOL;
    R103_1_I_RB_공기압_이상 AT %MW84102.9 : BOOL;
    R103_1_I_RB_냉각수_이상 AT %MW84102.10 : BOOL;
    R103_1_I_RB_비상정지_NC AT %MW84100.8 : BOOL;
    R103_1_I_RB_비전이상 AT %MW84102.14 : BOOL;
    R103_1_I_RB_실러이상 AT %MW84102.13 : BOOL;
    R103_1_I_RB_용접카운터이상 AT %MW84102.15 : BOOL;
    R103_1_I_RB_용접타점수 AT %MW84105 : WORD;
    R103_1_I_RB_운전준비 AT %MW84100.3 : BOOL;
    R103_1_I_RB_원위치 AT %MW84100.0 : BOOL;
    R103_1_I_RB_이상리셋 AT %MW84100.2 : BOOL;
    R103_1_I_RB_자동 AT %MW84100.4 : BOOL;
    R103_1_I_RB_자동기동 AT %MW84100.5 : BOOL;
    R103_1_I_RB_최종_작업완료 AT %MW84100.1 : BOOL;
    R103_1_I_RB_통신이상 AT %MW84102.12 : BOOL;
    R103_1_M_DATA_삭제_PLS AT %MW9006.0 : BOOL; (* R103_1_M_DATA_삭제_PLS *)
    R103_1_M_DATA_삭제_SIGN AT %MW9006.1 : BOOL; (* R103_1_M_DATA_삭제_SIGN *)
    R103_1_M_DATA_삭제_완료 AT %MW9006.2 : BOOL; (* R103_1_M_DATA_삭제_완료 *)
    R103_1_M_DATA_전송_MEMO AT %MW9006.8 : BOOL; (* R103_1_M_DATA_전송_MEMO *)
    R103_1_M_DATA_전송_PLS AT %MW9006.9 : BOOL; (* R103_1_M_DATA_전송_PLS *)
    R103_1_M_DATA_전송_SIGN AT %MW9006.10 : BOOL; (* R103_1_M_DATA_전송_SIGN *)
    R103_1_M_DATA_전송_완료 AT %MW9006.11 : BOOL; (* R103_1_M_DATA_전송_완료 *)
    R103_1_M_I_RB_1차_작업완료 AT %MW20101.2 : BOOL;
    R103_1_M_I_RB_2차_작업완료 AT %MW20101.3 : BOOL;
    R103_1_M_I_RB_3차_작업완료 AT %MW20101.4 : BOOL;
    R103_1_M_I_RB_4차_작업완료 AT %MW20101.5 : BOOL;
    R103_1_M_I_RB_5차_작업완료 AT %MW20101.6 : BOOL;
    R103_1_M_I_RB_6차_작업완료 AT %MW20101.7 : BOOL;
    R103_1_M_I_RB_7차_작업완료 AT %MW20101.8 : BOOL;
    R103_1_M_I_RB_PAUSE_보조 AT %MW20100.5 : BOOL;
    R103_1_M_I_RB_PLC_RUN_CHK_이상 AT %MW20100.7 : BOOL;
    R103_1_M_I_RB_간섭무_1 AT %MW20102.0 : BOOL;
    R103_1_M_I_RB_간섭무_10 AT %MW20102.9 : BOOL;
    R103_1_M_I_RB_간섭무_11 AT %MW20102.10 : BOOL;
    R103_1_M_I_RB_간섭무_12 AT %MW20102.11 : BOOL;
    R103_1_M_I_RB_간섭무_2 AT %MW20102.1 : BOOL;
    R103_1_M_I_RB_간섭무_3 AT %MW20102.2 : BOOL;
    R103_1_M_I_RB_간섭무_4 AT %MW20102.3 : BOOL;
    R103_1_M_I_RB_간섭무_5 AT %MW20102.4 : BOOL;
    R103_1_M_I_RB_간섭무_6 AT %MW20102.5 : BOOL;
    R103_1_M_I_RB_간섭무_7 AT %MW20102.6 : BOOL;
    R103_1_M_I_RB_간섭무_8 AT %MW20102.7 : BOOL;
    R103_1_M_I_RB_간섭무_9 AT %MW20102.8 : BOOL;
    R103_1_M_I_RB_비상정지 AT %MW20100.4 : BOOL;
    R103_1_M_I_RB_운전준비 AT %MW20100.0 : BOOL;
    R103_1_M_I_RB_원위치 AT %MW20100.3 : BOOL;
    R103_1_M_I_RB_이상 AT %MW20100.2 : BOOL;
    R103_1_M_I_RB_자동 AT %MW20100.1 : BOOL;
    R103_1_M_I_RB_최종작업완료 AT %MW20101.0 : BOOL;
    R103_1_M_I_RB_프로그램_이상 AT %MW20100.6 : BOOL;
    R103_1_M_O_RB_1_CYCLE_SET AT %MW21100.3 : BOOL;
    R103_1_M_O_RB_1_CYCLE_리셋 AT %MW21100.4 : BOOL;
    R103_1_M_O_RB_1차_작업완료_리셋 AT %MW21102.0 : BOOL;
    R103_1_M_O_RB_2차_작업완료_리셋 AT %MW21102.1 : BOOL;
    R103_1_M_O_RB_2차_진입OK AT %MW21101.8 : BOOL;
    R103_1_M_O_RB_3차_작업완료_리셋 AT %MW21102.2 : BOOL;
    R103_1_M_O_RB_3차_진입OK AT %MW21101.9 : BOOL;
    R103_1_M_O_RB_4차_작업완료_리셋 AT %MW21102.3 : BOOL;
    R103_1_M_O_RB_4차_진입OK AT %MW21101.10 : BOOL;
    R103_1_M_O_RB_5차_작업완료_리셋 AT %MW21102.4 : BOOL;
    R103_1_M_O_RB_5차_진입OK AT %MW21101.11 : BOOL;
    R103_1_M_O_RB_6차_작업완료_리셋 AT %MW21102.5 : BOOL;
    R103_1_M_O_RB_6차_진입OK AT %MW21101.12 : BOOL;
    R103_1_M_O_RB_7차_작업완료_리셋 AT %MW21102.6 : BOOL;
    R103_1_M_O_RB_7차_진입OK AT %MW21101.13 : BOOL;
    R103_1_M_O_RB_ATD_OK AT %MW21100.6 : BOOL;
    R103_1_M_O_RB_PLT_10_진입OK AT %MW21103.10 : BOOL;
    R103_1_M_O_RB_PLT_11_진입OK AT %MW21103.11 : BOOL;
    R103_1_M_O_RB_PLT_12_진입OK AT %MW21103.12 : BOOL;
    R103_1_M_O_RB_PLT_1_진입OK AT %MW21103.1 : BOOL;
    R103_1_M_O_RB_PLT_2_진입OK AT %MW21103.2 : BOOL;
    R103_1_M_O_RB_PLT_3_진입OK AT %MW21103.3 : BOOL;
    R103_1_M_O_RB_PLT_4_진입OK AT %MW21103.4 : BOOL;
    R103_1_M_O_RB_PLT_5_진입OK AT %MW21103.5 : BOOL;
    R103_1_M_O_RB_PLT_6_진입OK AT %MW21103.6 : BOOL;
    R103_1_M_O_RB_PLT_7_진입OK AT %MW21103.7 : BOOL;
    R103_1_M_O_RB_PLT_8_진입OK AT %MW21103.8 : BOOL;
    R103_1_M_O_RB_PLT_9_진입OK AT %MW21103.9 : BOOL;
    R103_1_M_O_RB_PLT_카운터리셋_보조 AT %MW21100.10 : BOOL;
    R103_1_M_O_RB_RESTART_OK AT %MW21100.2 : BOOL;
    R103_1_M_O_RB_START_OK AT %MW21100.0 : BOOL;
    R103_1_M_O_RB_TEST_MODE_5000회 AT %MW21100.12 : BOOL;
    R103_1_M_O_RB_TIP_교체_시작 AT %MW21100.7 : BOOL;
    R103_1_M_O_RB_TIP_교체_완료 AT %MW21100.8 : BOOL;
    R103_1_M_O_RB_VIP_MODE AT %MW21100.11 : BOOL;
    R103_1_M_O_RB_냉각수_차단_요청 AT %MW21100.9 : BOOL;
    R103_1_M_O_RB_진입OK_AX차종 AT %MW21101.0 : BOOL;
    R103_1_M_O_RB_진입OK_B차종 AT %MW21101.1 : BOOL;
    R103_1_M_O_RB_진입OK_C차종 AT %MW21101.2 : BOOL;
    R103_1_M_O_RB_진입OK_D차종 AT %MW21101.3 : BOOL;
    R103_1_M_O_RB_진입OK_E차종 AT %MW21101.4 : BOOL;
    R103_1_M_O_RB_진입OK_F차종 AT %MW21101.5 : BOOL;
    R103_1_M_O_RB_진입OK_G차종 AT %MW21101.6 : BOOL;
    R103_1_M_O_RB_진입OK_H차종 AT %MW21101.7 : BOOL;
    R103_1_M_O_RB_최종_작업완료_리셋 AT %MW21100.5 : BOOL;
    R103_1_M_O_RB_프로그램_OK AT %MW21100.1 : BOOL;
    R103_1_M_RB_PROG_NO AT %MW20104 : WORD;
    R103_1_M_RB_통신이상 AT %MW2024.1 : BOOL;
    R103_1_M_SEQ AT %MW10120 : WORD; (* R103_1_M_SEQ *)
    R103_1_M_STN_차종_NONE AT %MW2002.3 : BOOL;
    R103_1_M_STN_차종_ON AT %MW2002.2 : BOOL;
    R103_1_M_VIN_NO_1_2 AT %MW10131 : WORD; (* R103_1_M_VIN_NO_1_2 *)
    R103_1_M_VIN_NO_3_4 AT %MW10132 : WORD; (* R103_1_M_VIN_NO_3_4 *)
    R103_1_M_VIN_NO_5_6 AT %MW10133 : WORD; (* R103_1_M_VIN_NO_5_6 *)
    R103_1_M_VIN_NO_7_8 AT %MW10134 : WORD; (* R103_1_M_VIN_NO_7_8 *)
    R103_1_M_VIN_NO_9_10 AT %MW10135 : WORD; (* R103_1_M_VIN_NO_9_10 *)
    R103_1_M_차종1_AX AT %MW10121.0 : BOOL; (* R103_1_M_차종1_AX *)
    R103_1_M_차종1_B AT %MW10121.1 : BOOL; (* R103_1_M_차종1_B *)
    R103_1_M_차종1_C AT %MW10121.2 : BOOL; (* R103_1_M_차종1_C *)
    R103_1_M_차종1_D AT %MW10121.3 : BOOL; (* R103_1_M_차종1_D *)
    R103_1_M_차종1_E AT %MW10121.4 : BOOL; (* R103_1_M_차종1_E *)
    R103_1_M_차종1_F AT %MW10121.5 : BOOL; (* R103_1_M_차종1_F *)
    R103_1_M_차종1_G AT %MW10121.6 : BOOL; (* R103_1_M_차종1_G *)
    R103_1_M_차종1_H AT %MW10121.7 : BOOL; (* R103_1_M_차종1_H *)
    R103_1_M_차종2_3DR AT %MW10121.8 : BOOL; (* R103_1_M_차종2_3DR *)
    R103_1_M_차종2_4DR AT %MW10121.9 : BOOL; (* R103_1_M_차종2_4DR *)
    R103_1_M_차종2_5DR AT %MW10121.10 : BOOL; (* R103_1_M_차종2_5DR *)
    R103_1_M_차종2_SP1 AT %MW10121.12 : BOOL; (* R103_1_M_차종2_SP1 *)
    R103_1_M_차종2_SP2 AT %MW10121.13 : BOOL; (* R103_1_M_차종2_SP2 *)
    R103_1_M_차종2_WGN AT %MW10121.11 : BOOL; (* R103_1_M_차종2_WGN *)
    R103_1_M_차종3_LHD AT %MW10121.14 : BOOL; (* R103_1_M_차종3_LHD *)
    R103_1_M_차종3_RHD AT %MW10121.15 : BOOL; (* R103_1_M_차종3_RHD *)
    R103_1_M_차종4_EEC AT %MW10122.3 : BOOL; (* R103_1_M_차종4_EEC *)
    R103_1_M_차종4_SP1 AT %MW10122.8 : BOOL; (* R103_1_M_차종4_SP1 *)
    R103_1_M_차종4_SP2 AT %MW10122.9 : BOOL; (* R103_1_M_차종4_SP2 *)
    R103_1_M_차종4_SP3 AT %MW10122.11 : BOOL; (* R103_1_M_차종4_SP3 *)
    R103_1_M_차종4_SP4 AT %MW10122.12 : BOOL; (* R103_1_M_차종4_SP4 *)
    R103_1_M_차종4_SP5 AT %MW10122.13 : BOOL; (* R103_1_M_차종4_SP5 *)
    R103_1_M_차종4_SP6 AT %MW10122.14 : BOOL; (* R103_1_M_차종4_SP6 *)
    R103_1_M_차종4_SP7 AT %MW10122.15 : BOOL; (* R103_1_M_차종4_SP7 *)
    R103_1_M_차종4_내수 AT %MW10122.0 : BOOL; (* R103_1_M_차종4_내수 *)
    R103_1_M_차종4_러시아 AT %MW10122.10 : BOOL; (* R103_1_M_차종4_러시아 *)
    R103_1_M_차종4_북미 AT %MW10122.2 : BOOL; (* R103_1_M_차종4_북미 *)
    R103_1_M_차종4_브라질 AT %MW10122.7 : BOOL; (* R103_1_M_차종4_브라질 *)
    R103_1_M_차종4_수출 AT %MW10122.1 : BOOL; (* R103_1_M_차종4_수출 *)
    R103_1_M_차종4_중국 AT %MW10122.6 : BOOL; (* R103_1_M_차종4_중국 *)
    R103_1_M_차종4_중동 AT %MW10122.5 : BOOL; (* R103_1_M_차종4_중동 *)
    R103_1_M_차종4_호주 AT %MW10122.4 : BOOL; (* R103_1_M_차종4_호주 *)
    R103_1_M_차종5_AT AT %MW10123.1 : BOOL; (* R103_1_M_차종5_AT *)
    R103_1_M_차종5_MT AT %MW10123.0 : BOOL; (* R103_1_M_차종5_MT *)
    R103_1_M_차종5_SP1 AT %MW10123.2 : BOOL; (* R103_1_M_차종5_SP1 *)
    R103_1_M_차종6_DSROOF AT %MW10123.6 : BOOL; (* R103_1_M_차종6_DSROOF *)
    R103_1_M_차종6_SP1 AT %MW10123.7 : BOOL; (* R103_1_M_차종6_SP1 *)
    R103_1_M_차종6_썬루프 AT %MW10123.4 : BOOL; (* R103_1_M_차종6_썬루프 *)
    R103_1_M_차종6_일반루프 AT %MW10123.3 : BOOL; (* R103_1_M_차종6_일반루프 *)
    R103_1_M_차종6_파노라마루프 AT %MW10123.5 : BOOL; (* R103_1_M_차종6_파노라마루프 *)
    R103_1_M_차종7_DSL AT %MW10123.9 : BOOL; (* R103_1_M_차종7_DSL *)
    R103_1_M_차종7_GSL AT %MW10123.8 : BOOL; (* R103_1_M_차종7_GSL *)
    R103_1_M_차종7_SP1 AT %MW10123.10 : BOOL; (* R103_1_M_차종7_SP1 *)
    R103_1_M_차종7_SP2 AT %MW10123.11 : BOOL; (* R103_1_M_차종7_SP2 *)
    R103_1_M_차종7_SP3 AT %MW10123.12 : BOOL; (* R103_1_M_차종7_SP3 *)
    R103_1_M_차종7_SP4 AT %MW10123.13 : BOOL; (* R103_1_M_차종7_SP4 *)
    R103_1_M_차종7_SP5 AT %MW10123.14 : BOOL; (* R103_1_M_차종7_SP5 *)
    R103_1_M_차종7_SP6 AT %MW10123.15 : BOOL; (* R103_1_M_차종7_SP6 *)
    R103_1_M_차종8_2WD AT %MW10124.0 : BOOL; (* R103_1_M_차종8_2WD *)
    R103_1_M_차종8_4WD AT %MW10124.1 : BOOL; (* R103_1_M_차종8_4WD *)
    R103_1_M_차종8_SP1 AT %MW10124.2 : BOOL; (* R103_1_M_차종8_SP1 *)
    R103_1_M_차종9_MPI AT %MW10124.3 : BOOL; (* R103_1_M_차종9_MPI *)
    R103_1_M_차종9_SP1 AT %MW10124.5 : BOOL; (* R103_1_M_차종9_SP1 *)
    R103_1_M_차종9_SP10 AT %MW10124.14 : BOOL; (* R103_1_M_차종9_SP10 *)
    R103_1_M_차종9_SP11 AT %MW10124.15 : BOOL; (* R103_1_M_차종9_SP11 *)
    R103_1_M_차종9_SP2 AT %MW10124.6 : BOOL; (* R103_1_M_차종9_SP2 *)
    R103_1_M_차종9_SP3 AT %MW10124.7 : BOOL; (* R103_1_M_차종9_SP3 *)
    R103_1_M_차종9_SP4 AT %MW10124.8 : BOOL; (* R103_1_M_차종9_SP4 *)
    R103_1_M_차종9_SP5 AT %MW10124.9 : BOOL; (* R103_1_M_차종9_SP5 *)
    R103_1_M_차종9_SP6 AT %MW10124.10 : BOOL; (* R103_1_M_차종9_SP6 *)
    R103_1_M_차종9_SP7 AT %MW10124.11 : BOOL; (* R103_1_M_차종9_SP7 *)
    R103_1_M_차종9_SP8 AT %MW10124.12 : BOOL; (* R103_1_M_차종9_SP8 *)
    R103_1_M_차종9_SP9 AT %MW10124.13 : BOOL; (* R103_1_M_차종9_SP9 *)
    R103_1_M_차종9_T_GDI AT %MW10124.4 : BOOL; (* R103_1_M_차종9_T_GDI *)
    R103_1_M_차종_AS AT %MW10130.9 : BOOL; (* R103_1_M_차종_AS *)
    R103_1_M_차종_OPT1_R_RACK_무 AT %MW10125.3 : BOOL; (* R103_1_M_차종_OPT1_R_RACK_무 *)
    R103_1_M_차종_OPT1_R_RACK_유 AT %MW10125.2 : BOOL; (* R103_1_M_차종_OPT1_R_RACK_유 *)
    R103_1_M_차종_OPT1_SP1 AT %MW10125.10 : BOOL; (* R103_1_M_차종_OPT1_SP1 *)
    R103_1_M_차종_OPT1_SP2 AT %MW10125.11 : BOOL; (* R103_1_M_차종_OPT1_SP2 *)
    R103_1_M_차종_OPT1_SP3 AT %MW10125.12 : BOOL; (* R103_1_M_차종_OPT1_SP3 *)
    R103_1_M_차종_OPT1_SP4 AT %MW10125.13 : BOOL; (* R103_1_M_차종_OPT1_SP4 *)
    R103_1_M_차종_OPT1_SP5 AT %MW10125.14 : BOOL; (* R103_1_M_차종_OPT1_SP5 *)
    R103_1_M_차종_OPT1_SP6 AT %MW10125.15 : BOOL; (* R103_1_M_차종_OPT1_SP6 *)
    R103_1_M_차종_OPT1_S_REP_EATER_무 AT %MW10125.7 : BOOL; (* R103_1_M_차종_OPT1_S_REP_EATER_무 *)
    R103_1_M_차종_OPT1_S_REP_EATER_유 AT %MW10125.6 : BOOL; (* R103_1_M_차종_OPT1_S_REP_EATER_유 *)
    R103_1_M_차종_OPT1_VAN_무 AT %MW10125.9 : BOOL; (* R103_1_M_차종_OPT1_VAN_무 *)
    R103_1_M_차종_OPT1_VAN_유 AT %MW10125.8 : BOOL; (* R103_1_M_차종_OPT1_VAN_유 *)
    R103_1_M_차종_OPT1_슬라이딩_무 AT %MW10125.1 : BOOL; (* R103_1_M_차종_OPT1_슬라이딩_무 *)
    R103_1_M_차종_OPT1_슬라이딩_유 AT %MW10125.0 : BOOL; (* R103_1_M_차종_OPT1_슬라이딩_유 *)
    R103_1_M_차종_OPT1_폴딩_무 AT %MW10125.5 : BOOL; (* R103_1_M_차종_OPT1_폴딩_무 *)
    R103_1_M_차종_OPT1_폴딩_유 AT %MW10125.4 : BOOL; (* R103_1_M_차종_OPT1_폴딩_유 *)
    R103_1_M_차종_OPT2_SP_WORD1 AT %MW10126 : WORD; (* R103_1_M_차종_OPT2_SP_WORD1 *)
    R103_1_M_차종_OPT3_SP_WORD2 AT %MW10127 : WORD; (* R103_1_M_차종_OPT3_SP_WORD2 *)
    R103_1_M_차종_OPT4_SP_WORD3 AT %MW10128 : WORD; (* R103_1_M_차종_OPT4_SP_WORD3 *)
    R103_1_M_차종_OPT5_SP_WORD4 AT %MW10129 : WORD; (* R103_1_M_차종_OPT5_SP_WORD4 *)
    R103_1_M_차종_SP1 AT %MW10130.0 : BOOL; (* R103_1_M_차종_SP1 *)
    R103_1_M_차종_SP2 AT %MW10130.1 : BOOL; (* R103_1_M_차종_SP2 *)
    R103_1_M_차종_SP3 AT %MW10130.2 : BOOL; (* R103_1_M_차종_SP3 *)
    R103_1_M_차종_SP4 AT %MW10130.3 : BOOL; (* R103_1_M_차종_SP4 *)
    R103_1_M_차종_SP5 AT %MW10130.4 : BOOL; (* R103_1_M_차종_SP5 *)
    R103_1_M_차종_SP6 AT %MW10130.5 : BOOL; (* R103_1_M_차종_SP6 *)
    R103_1_M_차종_SP7 AT %MW10130.6 : BOOL; (* R103_1_M_차종_SP7 *)
    R103_1_M_차종_SP8 AT %MW10130.7 : BOOL; (* R103_1_M_차종_SP8 *)
    R103_1_M_차종_SP9 AT %MW10130.15 : BOOL; (* R103_1_M_차종_SP9 *)
    R103_1_M_차종_공대차 AT %MW10130.12 : BOOL; (* R103_1_M_차종_공대차 *)
    R103_1_M_차종_공차 AT %MW10130.10 : BOOL; (* R103_1_M_차종_공차 *)
    R103_1_M_차종_불량대차 AT %MW10130.13 : BOOL; (* R103_1_M_차종_불량대차 *)
    R103_1_M_차종_불량차 AT %MW10130.11 : BOOL; (* R103_1_M_차종_불량차 *)
    R103_1_M_차종_비축 AT %MW10130.8 : BOOL; (* R103_1_M_차종_비축 *)
    R103_1_M_차종_취출대차 AT %MW10130.14 : BOOL; (* R103_1_M_차종_취출대차 *)
    R103_1_O_RB_0_5S_통신_CHK AT %MW94103.14 : BOOL;
    R103_1_O_RB_2차_진입OK AT %MW94101.8 : BOOL;
    R103_1_O_RB_3차_진입OK AT %MW94101.9 : BOOL;
    R103_1_O_RB_4차_진입OK AT %MW94101.10 : BOOL;
    R103_1_O_RB_5차_진입OK AT %MW94101.11 : BOOL;
    R103_1_O_RB_6차_진입OK AT %MW94101.12 : BOOL;
    R103_1_O_RB_7차_진입OK AT %MW94101.13 : BOOL;
    R103_1_O_RB_AX_1차_진입OK AT %MW94101.0 : BOOL;
    R103_1_O_RB_B_1차_진입OK AT %MW94101.1 : BOOL;
    R103_1_O_RB_C_1차_진입OK AT %MW94101.2 : BOOL;
    R103_1_O_RB_D_1차_진입OK AT %MW94101.3 : BOOL;
    R103_1_O_RB_EACH_작업완료_리셋 AT %MW94100.14 : BOOL;
    R103_1_O_RB_EXT_READY AT %MW94100.11 : BOOL;
    R103_1_O_RB_E_1차_진입OK AT %MW94101.4 : BOOL;
    R103_1_O_RB_F_1차_진입OK AT %MW94101.5 : BOOL;
    R103_1_O_RB_GATE_OPEN_NC AT %MW94103.11 : BOOL;
    R103_1_O_RB_G_1차_진입OK AT %MW94101.6 : BOOL;
    R103_1_O_RB_H_1차_진입OK AT %MW94101.7 : BOOL;
    R103_1_O_RB_MUTUAL_INT1 AT %MW94103.0 : BOOL;
    R103_1_O_RB_MUTUAL_INT2 AT %MW94103.1 : BOOL;
    R103_1_O_RB_MUTUAL_INT3 AT %MW94103.2 : BOOL;
    R103_1_O_RB_MUTUAL_INT4 AT %MW94103.3 : BOOL;
    R103_1_O_RB_MUTUAL_INT5 AT %MW94103.4 : BOOL;
    R103_1_O_RB_MUTUAL_INT6 AT %MW94103.5 : BOOL;
    R103_1_O_RB_MUTUAL_INT7 AT %MW94103.6 : BOOL;
    R103_1_O_RB_MUTUAL_INT8 AT %MW94103.7 : BOOL;
    R103_1_O_RB_OUTPUT AT %MW94100 : ARRAY[0..3] OF WORD;
    R103_1_O_RB_PAUSE_NC AT %MW94100.13 : BOOL;
    R103_1_O_RB_PLT10_진입OK AT %MW94102.9 : BOOL;
    R103_1_O_RB_PLT11_진입OK AT %MW94102.10 : BOOL;
    R103_1_O_RB_PLT12_진입OK AT %MW94102.11 : BOOL;
    R103_1_O_RB_PLT1_진입OK AT %MW94102.0 : BOOL;
    R103_1_O_RB_PLT2_진입OK AT %MW94102.1 : BOOL;
    R103_1_O_RB_PLT3_진입OK AT %MW94102.2 : BOOL;
    R103_1_O_RB_PLT4_진입OK AT %MW94102.3 : BOOL;
    R103_1_O_RB_PLT5_진입OK AT %MW94102.4 : BOOL;
    R103_1_O_RB_PLT6_진입OK AT %MW94102.5 : BOOL;
    R103_1_O_RB_PLT7_진입OK AT %MW94102.6 : BOOL;
    R103_1_O_RB_PLT8_진입OK AT %MW94102.7 : BOOL;
    R103_1_O_RB_PLT9_진입OK AT %MW94102.8 : BOOL;
    R103_1_O_RB_PLT_COUNT_리셋_COND AT %MW94103.10 : BOOL;
    R103_1_O_RB_PROG_선택1 AT %MW94100.0 : BOOL;
    R103_1_O_RB_PROG_선택128 AT %MW94100.7 : BOOL;
    R103_1_O_RB_PROG_선택16 AT %MW94100.4 : BOOL;
    R103_1_O_RB_PROG_선택2 AT %MW94100.1 : BOOL;
    R103_1_O_RB_PROG_선택32 AT %MW94100.5 : BOOL;
    R103_1_O_RB_PROG_선택4 AT %MW94100.2 : BOOL;
    R103_1_O_RB_PROG_선택64 AT %MW94100.6 : BOOL;
    R103_1_O_RB_PROG_선택8 AT %MW94100.3 : BOOL;
    R103_1_O_RB_SP_1_14 AT %MW94101.14 : BOOL;
    R103_1_O_RB_SP_1_15 AT %MW94101.15 : BOOL;
    R103_1_O_RB_SP_2_12 AT %MW94102.12 : BOOL;
    R103_1_O_RB_SP_2_13 AT %MW94102.13 : BOOL;
    R103_1_O_RB_SP_2_14 AT %MW94102.14 : BOOL;
    R103_1_O_RB_SP_5000TH_ON AT %MW94102.15 : BOOL;
    R103_1_O_RB_TIP_CHANGE_END AT %MW94103.9 : BOOL;
    R103_1_O_RB_TIP_CHANGE_START AT %MW94103.8 : BOOL;
    R103_1_O_RB_TIP_DRESS_SATRT AT %MW94100.12 : BOOL;
    R103_1_O_RB_VIP_MODE AT %MW94103.15 : BOOL;
    R103_1_O_RB_기동 AT %MW94100.9 : BOOL;
    R103_1_O_RB_냉각수차단 AT %MW94100.15 : BOOL;
    R103_1_O_RB_부저정지 AT %MW94103.13 : BOOL;
    R103_1_O_RB_비상정지_NC AT %MW94103.12 : BOOL;
    R103_1_O_RB_이상_리셋 AT %MW94100.10 : BOOL;
    R103_1_O_RB_작업완료_리셋 AT %MW94100.8 : BOOL;
    R161_1_M_I_RB_1차_작업완료 AT %MW20111.2 : BOOL;
    R161_1_M_I_RB_최종작업완료 AT %MW20111.0 : BOOL;
    R161_1_M_O_RB_1차_작업완료_리셋 AT %MW21112.0 : BOOL;
    R161_1_M_O_RB_최종_작업완료_리셋 AT %MW21110.5 : BOOL;
    R161_2_M_I_RB_1차_작업완료 AT %MW20121.2 : BOOL;
    R161_2_M_I_RB_최종작업완료 AT %MW20121.0 : BOOL;
    R161_2_M_O_RB_1차_작업완료_리셋 AT %MW21122.0 : BOOL;
    R161_2_M_O_RB_최종_작업완료_리셋 AT %MW21120.5 : BOOL;
    R161_3축_리어_M_I_RB_1차_작업완료 AT %MW20191.2 : BOOL;
    R161_3축_리어_M_I_RB_2차_작업완료 AT %MW20191.3 : BOOL;
    R161_3축_리어_M_I_RB_3차_작업완료 AT %MW20191.4 : BOOL;
    R161_3축_리어_M_I_RB_4차_작업완료 AT %MW20191.5 : BOOL;
    R161_3축_리어_M_I_RB_5차_작업완료 AT %MW20191.6 : BOOL;
    R161_3축_리어_M_I_RB_6차_작업완료 AT %MW20191.7 : BOOL;
    R161_3축_리어_M_I_RB_7차_작업완료 AT %MW20191.8 : BOOL;
    R161_3축_리어_M_I_RB_PAUSE_보조 AT %MW20190.5 : BOOL;
    R161_3축_리어_M_I_RB_PLC_운전_CHK_이상 AT %MW20190.7 : BOOL;
    R161_3축_리어_M_I_RB_간섭무_1 AT %MW20192.0 : BOOL;
    R161_3축_리어_M_I_RB_간섭무_10 AT %MW20192.9 : BOOL;
    R161_3축_리어_M_I_RB_간섭무_11 AT %MW20192.10 : BOOL;
    R161_3축_리어_M_I_RB_간섭무_12 AT %MW20192.11 : BOOL;
    R161_3축_리어_M_I_RB_간섭무_2 AT %MW20192.1 : BOOL;
    R161_3축_리어_M_I_RB_간섭무_3 AT %MW20192.2 : BOOL;
    R161_3축_리어_M_I_RB_간섭무_4 AT %MW20192.3 : BOOL;
    R161_3축_리어_M_I_RB_간섭무_5 AT %MW20192.4 : BOOL;
    R161_3축_리어_M_I_RB_간섭무_6 AT %MW20192.5 : BOOL;
    R161_3축_리어_M_I_RB_간섭무_7 AT %MW20192.6 : BOOL;
    R161_3축_리어_M_I_RB_간섭무_8 AT %MW20192.7 : BOOL;
    R161_3축_리어_M_I_RB_간섭무_9 AT %MW20192.8 : BOOL;
    R161_3축_리어_M_I_RB_비상정지 AT %MW20190.4 : BOOL;
    R161_3축_리어_M_I_RB_운전준비 AT %MW20190.0 : BOOL;
    R161_3축_리어_M_I_RB_원위치 AT %MW20190.3 : BOOL;
    R161_3축_리어_M_I_RB_이상 AT %MW20190.2 : BOOL;
    R161_3축_리어_M_I_RB_자동 AT %MW20190.1 : BOOL;
    R161_3축_리어_M_I_RB_최종작업완료 AT %MW20191.0 : BOOL;
    R161_3축_리어_M_I_RB_프로그램_이상 AT %MW20190.6 : BOOL;
    R161_3축_리어_M_O_RB_1_CYCLE_SET AT %MW21190.3 : BOOL;
    R161_3축_리어_M_O_RB_1차_작업완료_리셋 AT %MW21192.0 : BOOL;
    R161_3축_리어_M_O_RB_2차_작업완료_리셋 AT %MW21192.1 : BOOL;
    R161_3축_리어_M_O_RB_2차_진입OK AT %MW21191.8 : BOOL;
    R161_3축_리어_M_O_RB_3차_작업완료_리셋 AT %MW21192.2 : BOOL;
    R161_3축_리어_M_O_RB_3차_진입OK AT %MW21191.9 : BOOL;
    R161_3축_리어_M_O_RB_4차_작업완료_리셋 AT %MW21192.3 : BOOL;
    R161_3축_리어_M_O_RB_4차_진입OK AT %MW21191.10 : BOOL;
    R161_3축_리어_M_O_RB_5차_작업완료_리셋 AT %MW21192.4 : BOOL;
    R161_3축_리어_M_O_RB_5차_진입OK AT %MW21191.11 : BOOL;
    R161_3축_리어_M_O_RB_6차_작업완료_리셋 AT %MW21192.5 : BOOL;
    R161_3축_리어_M_O_RB_6차_진입OK AT %MW21191.12 : BOOL;
    R161_3축_리어_M_O_RB_7차_작업완료_리셋 AT %MW21192.6 : BOOL;
    R161_3축_리어_M_O_RB_7차_진입OK AT %MW21191.13 : BOOL;
    R161_3축_리어_M_O_RB_ATD_OK AT %MW21190.6 : BOOL;
    R161_3축_리어_M_O_RB_PLT_10_진입OK AT %MW21193.10 : BOOL;
    R161_3축_리어_M_O_RB_PLT_11_진입OK AT %MW21193.11 : BOOL;
    R161_3축_리어_M_O_RB_PLT_12_진입OK AT %MW21193.12 : BOOL;
    R161_3축_리어_M_O_RB_PLT_1_진입OK AT %MW21193.1 : BOOL;
    R161_3축_리어_M_O_RB_PLT_2_진입OK AT %MW21193.2 : BOOL;
    R161_3축_리어_M_O_RB_PLT_3_진입OK AT %MW21193.3 : BOOL;
    R161_3축_리어_M_O_RB_PLT_4_진입OK AT %MW21193.4 : BOOL;
    R161_3축_리어_M_O_RB_PLT_5_진입OK AT %MW21193.5 : BOOL;
    R161_3축_리어_M_O_RB_PLT_6_진입OK AT %MW21193.6 : BOOL;
    R161_3축_리어_M_O_RB_PLT_7_진입OK AT %MW21193.7 : BOOL;
    R161_3축_리어_M_O_RB_PLT_8_진입OK AT %MW21193.8 : BOOL;
    R161_3축_리어_M_O_RB_PLT_9_진입OK AT %MW21193.9 : BOOL;
    R161_3축_리어_M_O_RB_PLT_카운터리셋_보조 AT %MW21190.10 : BOOL;
    R161_3축_리어_M_O_RB_RESTART_OK AT %MW21190.2 : BOOL;
    R161_3축_리어_M_O_RB_START_OK AT %MW21190.0 : BOOL;
    R161_3축_리어_M_O_RB_TEST_모드_5000회 AT %MW21190.12 : BOOL;
    R161_3축_리어_M_O_RB_TIP_교체_시작 AT %MW21190.7 : BOOL;
    R161_3축_리어_M_O_RB_TIP_교체_완료 AT %MW21190.8 : BOOL;
    R161_3축_리어_M_O_RB_VIP_모드 AT %MW21190.11 : BOOL;
    R161_3축_리어_M_O_RB_냉각수_차단_요청 AT %MW21190.9 : BOOL;
    R161_3축_리어_M_O_RB_진입OK_AX차종 AT %MW21191.0 : BOOL;
    R161_3축_리어_M_O_RB_진입OK_B차종 AT %MW21191.1 : BOOL;
    R161_3축_리어_M_O_RB_진입OK_C차종 AT %MW21191.2 : BOOL;
    R161_3축_리어_M_O_RB_진입OK_D차종 AT %MW21191.3 : BOOL;
    R161_3축_리어_M_O_RB_진입OK_E차종 AT %MW21191.4 : BOOL;
    R161_3축_리어_M_O_RB_진입OK_F차종 AT %MW21191.5 : BOOL;
    R161_3축_리어_M_O_RB_진입OK_G차종 AT %MW21191.6 : BOOL;
    R161_3축_리어_M_O_RB_진입OK_H차종 AT %MW21191.7 : BOOL;
    R161_3축_리어_M_O_RB_최종_작업완료_리셋 AT %MW21190.5 : BOOL;
    R161_3축_리어_M_O_RB_프로그램_OK AT %MW21190.1 : BOOL;
    R161_3축_리어_O_RB_OUTPUT AT %MW94190 : ARRAY[0..3] OF WORD;
    R161_3축_센터_I_RB_INPUT AT %MW84180 : ARRAY[0..3] OF WORD;
    R161_3축_센터_M_I_RB_1차_작업완료 AT %MW20181.2 : BOOL;
    R161_3축_센터_M_I_RB_2차_작업완료 AT %MW20181.3 : BOOL;
    R161_3축_센터_M_I_RB_3차_작업완료 AT %MW20181.4 : BOOL;
    R161_3축_센터_M_I_RB_4차_작업완료 AT %MW20181.5 : BOOL;
    R161_3축_센터_M_I_RB_5차_작업완료 AT %MW20181.6 : BOOL;
    R161_3축_센터_M_I_RB_6차_작업완료 AT %MW20181.7 : BOOL;
    R161_3축_센터_M_I_RB_7차_작업완료 AT %MW20181.8 : BOOL;
    R161_3축_센터_M_I_RB_PAUSE_보조 AT %MW20180.5 : BOOL;
    R161_3축_센터_M_I_RB_PLC_운전_CHK_이상 AT %MW20180.7 : BOOL;
    R161_3축_센터_M_I_RB_간섭무_1 AT %MW20182.0 : BOOL;
    R161_3축_센터_M_I_RB_간섭무_10 AT %MW20182.9 : BOOL;
    R161_3축_센터_M_I_RB_간섭무_11 AT %MW20182.10 : BOOL;
    R161_3축_센터_M_I_RB_간섭무_12 AT %MW20182.11 : BOOL;
    R161_3축_센터_M_I_RB_간섭무_2 AT %MW20182.1 : BOOL;
    R161_3축_센터_M_I_RB_간섭무_3 AT %MW20182.2 : BOOL;
    R161_3축_센터_M_I_RB_간섭무_4 AT %MW20182.3 : BOOL;
    R161_3축_센터_M_I_RB_간섭무_5 AT %MW20182.4 : BOOL;
    R161_3축_센터_M_I_RB_간섭무_6 AT %MW20182.5 : BOOL;
    R161_3축_센터_M_I_RB_간섭무_7 AT %MW20182.6 : BOOL;
    R161_3축_센터_M_I_RB_간섭무_8 AT %MW20182.7 : BOOL;
    R161_3축_센터_M_I_RB_간섭무_9 AT %MW20182.8 : BOOL;
    R161_3축_센터_M_I_RB_비상정지 AT %MW20180.4 : BOOL;
    R161_3축_센터_M_I_RB_운전준비 AT %MW20180.0 : BOOL;
    R161_3축_센터_M_I_RB_원위치 AT %MW20180.3 : BOOL;
    R161_3축_센터_M_I_RB_이상 AT %MW20180.2 : BOOL;
    R161_3축_센터_M_I_RB_자동 AT %MW20180.1 : BOOL;
    R161_3축_센터_M_I_RB_최종작업완료 AT %MW20181.0 : BOOL;
    R161_3축_센터_M_I_RB_프로그램_이상 AT %MW20180.6 : BOOL;
    R161_3축_센터_M_O_RB_1_CYCLE_SET AT %MW21180.3 : BOOL;
    R161_3축_센터_M_O_RB_1차_작업완료_리셋 AT %MW21182.0 : BOOL;
    R161_3축_센터_M_O_RB_2차_작업완료_리셋 AT %MW21182.1 : BOOL;
    R161_3축_센터_M_O_RB_2차_진입OK AT %MW21181.8 : BOOL;
    R161_3축_센터_M_O_RB_3차_작업완료_리셋 AT %MW21182.2 : BOOL;
    R161_3축_센터_M_O_RB_3차_진입OK AT %MW21181.9 : BOOL;
    R161_3축_센터_M_O_RB_4차_작업완료_리셋 AT %MW21182.3 : BOOL;
    R161_3축_센터_M_O_RB_4차_진입OK AT %MW21181.10 : BOOL;
    R161_3축_센터_M_O_RB_5차_작업완료_리셋 AT %MW21182.4 : BOOL;
    R161_3축_센터_M_O_RB_5차_진입OK AT %MW21181.11 : BOOL;
    R161_3축_센터_M_O_RB_6차_작업완료_리셋 AT %MW21182.5 : BOOL;
    R161_3축_센터_M_O_RB_6차_진입OK AT %MW21181.12 : BOOL;
    R161_3축_센터_M_O_RB_7차_작업완료_리셋 AT %MW21182.6 : BOOL;
    R161_3축_센터_M_O_RB_7차_진입OK AT %MW21181.13 : BOOL;
    R161_3축_센터_M_O_RB_ATD_OK AT %MW21180.6 : BOOL;
    R161_3축_센터_M_O_RB_PLT_10_진입OK AT %MW21183.10 : BOOL;
    R161_3축_센터_M_O_RB_PLT_11_진입OK AT %MW21183.11 : BOOL;
    R161_3축_센터_M_O_RB_PLT_12_진입OK AT %MW21183.12 : BOOL;
    R161_3축_센터_M_O_RB_PLT_1_진입OK AT %MW21183.1 : BOOL;
    R161_3축_센터_M_O_RB_PLT_2_진입OK AT %MW21183.2 : BOOL;
    R161_3축_센터_M_O_RB_PLT_3_진입OK AT %MW21183.3 : BOOL;
    R161_3축_센터_M_O_RB_PLT_4_진입OK AT %MW21183.4 : BOOL;
    R161_3축_센터_M_O_RB_PLT_5_진입OK AT %MW21183.5 : BOOL;
    R161_3축_센터_M_O_RB_PLT_6_진입OK AT %MW21183.6 : BOOL;
    R161_3축_센터_M_O_RB_PLT_7_진입OK AT %MW21183.7 : BOOL;
    R161_3축_센터_M_O_RB_PLT_8_진입OK AT %MW21183.8 : BOOL;
    R161_3축_센터_M_O_RB_PLT_9_진입OK AT %MW21183.9 : BOOL;
    R161_3축_센터_M_O_RB_PLT_카운터리셋_보조 AT %MW21180.10 : BOOL;
    R161_3축_센터_M_O_RB_RESTART_OK AT %MW21180.2 : BOOL;
    R161_3축_센터_M_O_RB_START_OK AT %MW21180.0 : BOOL;
    R161_3축_센터_M_O_RB_TEST_모드_5000회 AT %MW21180.12 : BOOL;
    R161_3축_센터_M_O_RB_TIP_교체_시작 AT %MW21180.7 : BOOL;
    R161_3축_센터_M_O_RB_TIP_교체_완료 AT %MW21180.8 : BOOL;
    R161_3축_센터_M_O_RB_VIP_모드 AT %MW21180.11 : BOOL;
    R161_3축_센터_M_O_RB_냉각수_차단_요청 AT %MW21180.9 : BOOL;
    R161_3축_센터_M_O_RB_진입OK_AX차종 AT %MW21181.0 : BOOL;
    R161_3축_센터_M_O_RB_진입OK_B차종 AT %MW21181.1 : BOOL;
    R161_3축_센터_M_O_RB_진입OK_C차종 AT %MW21181.2 : BOOL;
    R161_3축_센터_M_O_RB_진입OK_D차종 AT %MW21181.3 : BOOL;
    R161_3축_센터_M_O_RB_진입OK_E차종 AT %MW21181.4 : BOOL;
    R161_3축_센터_M_O_RB_진입OK_F차종 AT %MW21181.5 : BOOL;
    R161_3축_센터_M_O_RB_진입OK_G차종 AT %MW21181.6 : BOOL;
    R161_3축_센터_M_O_RB_진입OK_H차종 AT %MW21181.7 : BOOL;
    R161_3축_센터_M_O_RB_최종_작업완료_리셋 AT %MW21180.5 : BOOL;
    R161_3축_센터_M_O_RB_프로그램_OK AT %MW21180.1 : BOOL;
    R161_3축_센터_M_RB_PROG_NO : INT;
    R161_3축_센터_O_RB_OUTPUT AT %MW94180 : ARRAY[0..3] OF WORD;
    R161_3축_프론트_I_RB_INPUT AT %MW84170 : ARRAY[0..3] OF WORD;
    R161_3축_프론트_M_I_RB_1차_작업완료 AT %MW20171.2 : BOOL;
    R161_3축_프론트_M_I_RB_2차_작업완료 AT %MW20171.3 : BOOL;
    R161_3축_프론트_M_I_RB_3차_작업완료 AT %MW20171.4 : BOOL;
    R161_3축_프론트_M_I_RB_4차_작업완료 AT %MW20171.5 : BOOL;
    R161_3축_프론트_M_I_RB_5차_작업완료 AT %MW20171.6 : BOOL;
    R161_3축_프론트_M_I_RB_6차_작업완료 AT %MW20171.7 : BOOL;
    R161_3축_프론트_M_I_RB_7차_작업완료 AT %MW20171.8 : BOOL;
    R161_3축_프론트_M_I_RB_PAUSE_보조 AT %MW20170.5 : BOOL;
    R161_3축_프론트_M_I_RB_PLC_운전_CHK_이상 AT %MW20170.7 : BOOL;
    R161_3축_프론트_M_I_RB_간섭무_1 AT %MW20172.0 : BOOL;
    R161_3축_프론트_M_I_RB_간섭무_10 AT %MW20172.9 : BOOL;
    R161_3축_프론트_M_I_RB_간섭무_11 AT %MW20172.10 : BOOL;
    R161_3축_프론트_M_I_RB_간섭무_12 AT %MW20172.11 : BOOL;
    R161_3축_프론트_M_I_RB_간섭무_2 AT %MW20172.1 : BOOL;
    R161_3축_프론트_M_I_RB_간섭무_3 AT %MW20172.2 : BOOL;
    R161_3축_프론트_M_I_RB_간섭무_4 AT %MW20172.3 : BOOL;
    R161_3축_프론트_M_I_RB_간섭무_5 AT %MW20172.4 : BOOL;
    R161_3축_프론트_M_I_RB_간섭무_6 AT %MW20172.5 : BOOL;
    R161_3축_프론트_M_I_RB_간섭무_7 AT %MW20172.6 : BOOL;
    R161_3축_프론트_M_I_RB_간섭무_8 AT %MW20172.7 : BOOL;
    R161_3축_프론트_M_I_RB_간섭무_9 AT %MW20172.8 : BOOL;
    R161_3축_프론트_M_I_RB_비상정지 AT %MW20170.4 : BOOL;
    R161_3축_프론트_M_I_RB_운전준비 AT %MW20170.0 : BOOL;
    R161_3축_프론트_M_I_RB_원위치 AT %MW20170.3 : BOOL;
    R161_3축_프론트_M_I_RB_이상 AT %MW20170.2 : BOOL;
    R161_3축_프론트_M_I_RB_자동 AT %MW20170.1 : BOOL;
    R161_3축_프론트_M_I_RB_최종작업완료 AT %MW20171.0 : BOOL;
    R161_3축_프론트_M_I_RB_프로그램_이상 AT %MW20170.6 : BOOL;
    R161_3축_프론트_M_O_RB_1_CYCLE_SET AT %MW21170.3 : BOOL;
    R161_3축_프론트_M_O_RB_1차_작업완료_리셋 AT %MW21172.0 : BOOL;
    R161_3축_프론트_M_O_RB_2차_작업완료_리셋 AT %MW21172.1 : BOOL;
    R161_3축_프론트_M_O_RB_2차_진입OK AT %MW21171.8 : BOOL;
    R161_3축_프론트_M_O_RB_3차_작업완료_리셋 AT %MW21172.2 : BOOL;
    R161_3축_프론트_M_O_RB_3차_진입OK AT %MW21171.9 : BOOL;
    R161_3축_프론트_M_O_RB_4차_작업완료_리셋 AT %MW21172.3 : BOOL;
    R161_3축_프론트_M_O_RB_4차_진입OK AT %MW21171.10 : BOOL;
    R161_3축_프론트_M_O_RB_5차_작업완료_리셋 AT %MW21172.4 : BOOL;
    R161_3축_프론트_M_O_RB_5차_진입OK AT %MW21171.11 : BOOL;
    R161_3축_프론트_M_O_RB_6차_작업완료_리셋 AT %MW21172.5 : BOOL;
    R161_3축_프론트_M_O_RB_6차_진입OK AT %MW21171.12 : BOOL;
    R161_3축_프론트_M_O_RB_7차_작업완료_리셋 AT %MW21172.6 : BOOL;
    R161_3축_프론트_M_O_RB_7차_진입OK AT %MW21171.13 : BOOL;
    R161_3축_프론트_M_O_RB_ATD_OK AT %MW21170.6 : BOOL;
    R161_3축_프론트_M_O_RB_PLT_10_진입OK AT %MW21173.10 : BOOL;
    R161_3축_프론트_M_O_RB_PLT_11_진입OK AT %MW21173.11 : BOOL;
    R161_3축_프론트_M_O_RB_PLT_12_진입OK AT %MW21173.12 : BOOL;
    R161_3축_프론트_M_O_RB_PLT_1_진입OK AT %MW21173.1 : BOOL;
    R161_3축_프론트_M_O_RB_PLT_2_진입OK AT %MW21173.2 : BOOL;
    R161_3축_프론트_M_O_RB_PLT_3_진입OK AT %MW21173.3 : BOOL;
    R161_3축_프론트_M_O_RB_PLT_4_진입OK AT %MW21173.4 : BOOL;
    R161_3축_프론트_M_O_RB_PLT_5_진입OK AT %MW21173.5 : BOOL;
    R161_3축_프론트_M_O_RB_PLT_6_진입OK AT %MW21173.6 : BOOL;
    R161_3축_프론트_M_O_RB_PLT_7_진입OK AT %MW21173.7 : BOOL;
    R161_3축_프론트_M_O_RB_PLT_8_진입OK AT %MW21173.8 : BOOL;
    R161_3축_프론트_M_O_RB_PLT_9_진입OK AT %MW21173.9 : BOOL;
    R161_3축_프론트_M_O_RB_PLT_카운터리셋_보조 AT %MW21170.10 : BOOL;
    R161_3축_프론트_M_O_RB_RESTART_OK AT %MW21170.2 : BOOL;
    R161_3축_프론트_M_O_RB_START_OK AT %MW21170.0 : BOOL;
    R161_3축_프론트_M_O_RB_TEST_모드_5000회 AT %MW21170.12 : BOOL;
    R161_3축_프론트_M_O_RB_TIP_교체_시작 AT %MW21170.7 : BOOL;
    R161_3축_프론트_M_O_RB_TIP_교체_완료 AT %MW21170.8 : BOOL;
    R161_3축_프론트_M_O_RB_VIP_모드 AT %MW21170.11 : BOOL;
    R161_3축_프론트_M_O_RB_냉각수_차단_요청 AT %MW21170.9 : BOOL;
    R161_3축_프론트_M_O_RB_진입OK_AX차종 AT %MW21171.0 : BOOL;
    R161_3축_프론트_M_O_RB_진입OK_B차종 AT %MW21171.1 : BOOL;
    R161_3축_프론트_M_O_RB_진입OK_C차종 AT %MW21171.2 : BOOL;
    R161_3축_프론트_M_O_RB_진입OK_D차종 AT %MW21171.3 : BOOL;
    R161_3축_프론트_M_O_RB_진입OK_E차종 AT %MW21171.4 : BOOL;
    R161_3축_프론트_M_O_RB_진입OK_F차종 AT %MW21171.5 : BOOL;
    R161_3축_프론트_M_O_RB_진입OK_G차종 AT %MW21171.6 : BOOL;
    R161_3축_프론트_M_O_RB_진입OK_H차종 AT %MW21171.7 : BOOL;
    R161_3축_프론트_M_O_RB_최종_작업완료_리셋 AT %MW21170.5 : BOOL;
    R161_3축_프론트_M_O_RB_프로그램_OK AT %MW21170.1 : BOOL;
    R161_3축_프론트_O_RB_OUTPUT AT %MW94170 : ARRAY[0..3] OF WORD;
    R162_3축_프론트_M_I_RB_1차_작업완료 AT %MW20281.2 : BOOL;
    R163_3축_프론트_M_I_RB_1차_작업완료 AT %MW20381.2 : BOOL;
    R164_3축_프론트_M_I_RB_1차_작업완료 AT %MW20481.2 : BOOL;
    R165_3축_프론트_M_I_RB_1차_작업완료 AT %MW20581.2 : BOOL;
    R166_3축_프론트_M_I_RB_1차_작업완료 : BOOL;
    S101_3축_1_ABSOLUTE AT %MW51002.8 : BOOL;
    S101_3축_1_ACCEL AT %MW51009 : WORD;
    S101_3축_1_COAST_정지 AT %MW51000.1 : BOOL;
    S101_3축_1_DECEL AT %MW51010 : WORD;
    S101_3축_1_ENALBLE1 AT %MW51000.0 : BOOL;
    S101_3축_1_ENALBLE2 AT %MW51000.3 : BOOL;
    S101_3축_1_FAULT AT %MW50000.3 : BOOL;
    S101_3축_1_FAULT_NUM AT %MW50009 : WORD;
    S101_3축_1_HOME AT %MW51000.11 : BOOL;
    S101_3축_1_HOME_SET AT %MW50000.11 : BOOL;
    S101_3축_1_INTERME_정지 AT %MW51000.5 : BOOL;
    S101_3축_1_JOG_MOVING AT %MW50001.10 : BOOL;
    S101_3축_1_JOG_전진 AT %MW51000.8 : BOOL;
    S101_3축_1_JOG_후진 AT %MW51000.9 : BOOL;
    S101_3축_1_MDI_선택 AT %MW51001.15 : BOOL;
    S101_3축_1_MOVE_COMP AT %MW50000.10 : BOOL;
    S101_3축_1_OUT_VELOCITY1 AT %MW51007 : WORD;
    S101_3축_1_OUT_VELOCITY2 AT %MW51008 : WORD;
    S101_3축_1_OVERRIDE AT %MW51004 : WORD;
    S101_3축_1_PLC_CONTROL AT %MW51000.10 : BOOL;
    S101_3축_1_POSITION AT %MD255 : DINT;
    S101_3축_1_POSITION1 AT %MW50005 : WORD;
    S101_3축_1_POSITION2 AT %MW50006 : WORD;
    S101_3축_1_QUICK_정지 AT %MW51000.2 : BOOL;
    S101_3축_1_SOFT_LIMIT AT %MW51002.14 : BOOL;
    S101_3축_1_START1 AT %MW51000.4 : BOOL;
    S101_3축_1_START2 AT %MW51000.6 : BOOL;
    S101_3축_1_TARGET_POSITION AT %MD280 : DINT;
    S101_3축_1_TARGET_POSITION1 AT %MW51005 : WORD;
    S101_3축_1_TARGET_POSITION2 AT %MW51006 : WORD;
    S101_3축_1_TRACK_모드 AT %MW51002.0 : BOOL;
    S101_3축_1_VELOCITY1 AT %MW50007 : WORD;
    S101_3축_1_VELOCITY2 AT %MW50008 : WORD;
    S101_3축_1_운전준비1 AT %MW50000.0 : BOOL;
    S101_3축_1_운전준비2 AT %MW50000.1 : BOOL;
    S101_3축_1_운전준비_COMP AT %MW50000.2 : BOOL;
    S101_3축_1_이상_리셋 AT %MW51000.7 : BOOL;
    S101_3축_2_ABSOLUTE AT %MW51102.8 : BOOL;
    S101_3축_2_ACCEL AT %MW51109 : WORD;
    S101_3축_2_COAST_정지 AT %MW51100.1 : BOOL;
    S101_3축_2_DECEL AT %MW51110 : WORD;
    S101_3축_2_ENALBLE1 AT %MW51100.0 : BOOL;
    S101_3축_2_ENALBLE2 AT %MW51100.3 : BOOL;
    S101_3축_2_FAULT AT %MW50100.3 : BOOL;
    S101_3축_2_FAULT_NUM AT %MW50109 : WORD;
    S101_3축_2_HOME AT %MW51100.11 : BOOL;
    S101_3축_2_HOME_SET AT %MW50100.11 : BOOL;
    S101_3축_2_INTERME_정지 AT %MW51100.5 : BOOL;
    S101_3축_2_JOG_MOVING AT %MW50101.10 : BOOL;
    S101_3축_2_JOG_전진 AT %MW51100.8 : BOOL;
    S101_3축_2_JOG_후진 AT %MW51100.9 : BOOL;
    S101_3축_2_MDI_선택 AT %MW51101.15 : BOOL;
    S101_3축_2_MOVE_COMP AT %MW50100.10 : BOOL;
    S101_3축_2_OUT_VELOCITY1 AT %MW51107 : WORD;
    S101_3축_2_OUT_VELOCITY2 AT %MW51108 : WORD;
    S101_3축_2_OVERRIDE AT %MW51104 : WORD;
    S101_3축_2_PLC_CONTROL AT %MW51100.10 : BOOL;
    S101_3축_2_POSITION AT %MD260 : DINT;
    S101_3축_2_POSITION1 AT %MW50105 : WORD;
    S101_3축_2_POSITION2 AT %MW50106 : WORD;
    S101_3축_2_QUICK_정지 AT %MW51100.2 : BOOL;
    S101_3축_2_SOFT_LIMIT AT %MW51102.14 : BOOL;
    S101_3축_2_START1 AT %MW51100.4 : BOOL;
    S101_3축_2_START2 AT %MW51100.6 : BOOL;
    S101_3축_2_TARGET_POSITION AT %MD285 : DINT;
    S101_3축_2_TARGET_POSITION1 AT %MW51105 : WORD;
    S101_3축_2_TARGET_POSITION2 AT %MW51106 : WORD;
    S101_3축_2_TRACK_모드 AT %MW51102.0 : BOOL;
    S101_3축_2_VELOCITY1 AT %MW50107 : WORD;
    S101_3축_2_VELOCITY2 AT %MW50108 : WORD;
    S101_3축_2_운전준비1 AT %MW50100.0 : BOOL;
    S101_3축_2_운전준비2 AT %MW50100.1 : BOOL;
    S101_3축_2_운전준비_COMP AT %MW50100.2 : BOOL;
    S101_3축_2_이상_리셋 AT %MW51100.7 : BOOL;
    S101_3축_3_ABSOLUTE AT %MW51202.8 : BOOL;
    S101_3축_3_ACCEL AT %MW51209 : WORD;
    S101_3축_3_COAST_정지 AT %MW51200.1 : BOOL;
    S101_3축_3_DECEL AT %MW51210 : WORD;
    S101_3축_3_ENALBLE1 AT %MW51200.0 : BOOL;
    S101_3축_3_ENALBLE2 AT %MW51200.3 : BOOL;
    S101_3축_3_FAULT AT %MW50200.3 : BOOL;
    S101_3축_3_FAULT_NUM AT %MW50209 : WORD;
    S101_3축_3_HOME AT %MW51200.11 : BOOL;
    S101_3축_3_HOME_SET AT %MW50200.11 : BOOL;
    S101_3축_3_INTERME_정지 AT %MW51200.5 : BOOL;
    S101_3축_3_JOG_MOVING AT %MW50201.10 : BOOL;
    S101_3축_3_JOG_전진 AT %MW51200.8 : BOOL;
    S101_3축_3_JOG_후진 AT %MW51200.9 : BOOL;
    S101_3축_3_MDI_선택 AT %MW51201.15 : BOOL;
    S101_3축_3_MOVE_COMP AT %MW50200.10 : BOOL;
    S101_3축_3_OUT_VELOCITY1 AT %MW51207 : WORD;
    S101_3축_3_OUT_VELOCITY2 AT %MW51208 : WORD;
    S101_3축_3_OVERRIDE AT %MW51204 : WORD;
    S101_3축_3_PLC_CONTROL AT %MW51200.10 : BOOL;
    S101_3축_3_POSITION AT %MD265 : DINT;
    S101_3축_3_POSITION1 AT %MW50205 : WORD;
    S101_3축_3_POSITION2 AT %MW50206 : WORD;
    S101_3축_3_QUICK_정지 AT %MW51200.2 : BOOL;
    S101_3축_3_SOFT_LIMIT AT %MW51202.14 : BOOL;
    S101_3축_3_START1 AT %MW51200.4 : BOOL;
    S101_3축_3_START2 AT %MW51200.6 : BOOL;
    S101_3축_3_TARGET_POSITION AT %MD290 : DINT;
    S101_3축_3_TARGET_POSITION1 AT %MW51205 : WORD;
    S101_3축_3_TARGET_POSITION2 AT %MW51206 : WORD;
    S101_3축_3_TRACK_모드 AT %MW51202.0 : BOOL;
    S101_3축_3_VELOCITY1 AT %MW50207 : WORD;
    S101_3축_3_VELOCITY2 AT %MW50208 : WORD;
    S101_3축_3_운전준비1 AT %MW50200.0 : BOOL;
    S101_3축_3_운전준비2 AT %MW50200.1 : BOOL;
    S101_3축_3_운전준비_COMP AT %MW50200.2 : BOOL;
    S101_3축_3_이상_리셋 AT %MW51200.7 : BOOL;
    S101_6_10_PLC_BOX_CP_TRIP AT %MW86102.15 : BOOL; (* 입력 접점 15 *)
    S101_AX_래치 : ACT_6_CYL;
    S101_DASH_클램프 : ACT_6_CYL;
    S101_HOME AT %MW1048.0 : BOOL;
    S101_IN_3축_1_CONTROL AT %MB100000 : ARRAY[0..23] OF BYTE;
    S101_IN_3축_1_EXPEN AT %MB100024 : ARRAY[0..31] OF BYTE;
    S101_IN_3축_2_CONTROL AT %MB100200 : ARRAY[0..23] OF BYTE;
    S101_IN_3축_2_EXPEN AT %MB100224 : ARRAY[0..31] OF BYTE;
    S101_IN_3축_3_CONTROL AT %MB100400 : ARRAY[0..23] OF BYTE;
    S101_IN_3축_3_EXPEN AT %MB100424 : ARRAY[0..31] OF BYTE;
    S101_JOG_OFF AT %MW1048.5 : BOOL;
    S101_JOG_ON AT %MW1048.4 : BOOL;
    S101_LH_M_APRON_PLT1_COUNT_RST AT %MW1200.15 : BOOL;
    S101_LH_M_APRON_PLT1_FAULT AT %MW1200.6 : BOOL;
    S101_LH_M_APRON_PLT1_MATCH_OK AT %MW1200.5 : BOOL;
    S101_LH_M_APRON_PLT1_PART_ERR AT %MW1200.9 : BOOL;
    S101_LH_M_APRON_PLT1_PLT_NONE AT %MW1200.2 : BOOL;
    S101_LH_M_APRON_PLT1_PLT_ON AT %MW1200.1 : BOOL;
    S101_LH_M_APRON_PLT1_PROG_OK AT %MW1200.0 : BOOL;
    S101_LH_M_APRON_PLT1_UNMAT_ERR AT %MW1200.7 : BOOL;
    S101_LH_M_APRON_PLT1_로딩완료 AT %MW1200.10 : BOOL;
    S101_LH_M_APRON_PLT1_제품수량 AT %MW1224 : WORD;
    S101_LH_M_APRON_PLT1_차종100 AT %MW1200.11 : BOOL;
    S101_LH_M_APRON_PLT1_차종200 AT %MW1200.12 : BOOL;
    S101_LH_M_APRON_PLT1_차종300 AT %MW1200.13 : BOOL;
    S101_LH_M_APRON_PLT1_차종400 AT %MW1200.14 : BOOL;
    S101_LH_M_APRON_PLT1_차종유 AT %MW1200.8 : BOOL;
    S101_LH_M_APRON_PLT1_차종코드 AT %MW1216 : WORD;
    S101_LH_M_APRON_PLT1_파트무 AT %MW1200.4 : BOOL;
    S101_LH_M_APRON_PLT1_파트유 AT %MW1200.3 : BOOL;
    S101_LH_M_APRON_PLT2_COUNT_RST AT %MW1201.15 : BOOL;
    S101_LH_M_APRON_PLT2_FAULT AT %MW1201.6 : BOOL;
    S101_LH_M_APRON_PLT2_MATCH_OK AT %MW1201.5 : BOOL;
    S101_LH_M_APRON_PLT2_PART_ERR AT %MW1201.9 : BOOL;
    S101_LH_M_APRON_PLT2_PLT_NONE AT %MW1201.2 : BOOL;
    S101_LH_M_APRON_PLT2_PLT_ON AT %MW1201.1 : BOOL;
    S101_LH_M_APRON_PLT2_PROG_OK AT %MW1201.0 : BOOL;
    S101_LH_M_APRON_PLT2_UNMAT_ERR AT %MW1201.7 : BOOL;
    S101_LH_M_APRON_PLT2_로딩완료 AT %MW1201.10 : BOOL;
    S101_LH_M_APRON_PLT2_제품수량 AT %MW1225 : WORD;
    S101_LH_M_APRON_PLT2_차종100 AT %MW1201.11 : BOOL;
    S101_LH_M_APRON_PLT2_차종200 AT %MW1201.12 : BOOL;
    S101_LH_M_APRON_PLT2_차종300 AT %MW1201.13 : BOOL;
    S101_LH_M_APRON_PLT2_차종400 AT %MW1201.14 : BOOL;
    S101_LH_M_APRON_PLT2_차종유 AT %MW1201.8 : BOOL;
    S101_LH_M_APRON_PLT2_차종코드 AT %MW1217 : WORD;
    S101_LH_M_APRON_PLT2_파트무 AT %MW1201.4 : BOOL;
    S101_LH_M_APRON_PLT2_파트유 AT %MW1201.3 : BOOL;
    S101_LH_M_APRON_PLT3_제품수량 AT %MW1226 : WORD;
    S101_LH_M_APRON_PLT3_차종코드 AT %MW1218 : WORD;
    S101_LH_M_APRON_PLT4_제품수량 AT %MW1227 : WORD;
    S101_LH_M_APRON_PLT4_차종코드 AT %MW1219 : WORD;
    S101_LH_M_APRON_PLT5_제품수량 AT %MW1228 : WORD;
    S101_LH_M_APRON_PLT5_차종코드 AT %MW1220 : WORD;
    S101_LH_M_APRON_PLT6_제품수량 AT %MW1229 : WORD;
    S101_LH_M_APRON_PLT6_차종코드 AT %MW1221 : WORD;
    S101_LH_M_APRON_PLT7_제품수량 AT %MW1230 : WORD;
    S101_LH_M_APRON_PLT7_차종코드 AT %MW1222 : WORD;
    S101_LH_M_APRON_PLT8_제품수량 AT %MW1231 : WORD;
    S101_LH_M_APRON_PLT8_차종코드 AT %MW1223 : WORD;
    S101_LH_M_APRON_PLT_PRIORITY1 AT %MW1208 : WORD;
    S101_LH_M_APRON_PLT_PRIORITY2 AT %MW1209 : WORD;
    S101_LH_M_APRON_PLT_PRIORITY3 AT %MW1210 : WORD;
    S101_LH_M_APRON_PLT_PRIORITY4 AT %MW1211 : WORD;
    S101_LH_M_APRON_PLT_PRIORITY5 AT %MW1212 : WORD;
    S101_LH_M_APRON_PLT_PRIORITY6 AT %MW1213 : WORD;
    S101_LH_M_APRON_PLT_PRIORITY7 AT %MW1214 : WORD;
    S101_LH_M_APRON_PLT_PRIORITY8 AT %MW1215 : WORD;
    S101_MCR_비상정지1 AT %MW95207.0 : BOOL; (* 출력 접점 00 *)
    S101_MCR_비상정지2 AT %MW95207.1 : BOOL; (* 출력 접점 01 *)
    S101_MCR_비상정지3 AT %MW95207.2 : BOOL; (* 출력 접점 02 *)
    S101_M_3_축1_전진_LS_이상 AT %MW1102.5 : BOOL;
    S101_M_3_축1_전진_보조 AT %MW1102.1 : BOOL;
    S101_M_3_축1_전진단 AT %MW1102.3 : BOOL;
    S101_M_3_축1_조건 AT %MW1102.0 : BOOL;
    S101_M_3_축1_후진_LS_이상 AT %MW1102.6 : BOOL;
    S101_M_3_축1_후진_보조 AT %MW1102.2 : BOOL;
    S101_M_3_축1_후진단 AT %MW1102.4 : BOOL;
    S101_M_3_축2_전진_LS_이상 AT %MW1103.5 : BOOL;
    S101_M_3_축2_전진_보조 AT %MW1103.1 : BOOL;
    S101_M_3_축2_전진단 AT %MW1103.3 : BOOL;
    S101_M_3_축2_조건 AT %MW1103.0 : BOOL;
    S101_M_3_축2_후진_LS_이상 AT %MW1103.6 : BOOL;
    S101_M_3_축2_후진_보조 AT %MW1103.2 : BOOL;
    S101_M_3_축2_후진단 AT %MW1103.4 : BOOL;
    S101_M_3_축3_전진_LS_이상 AT %MW1104.5 : BOOL;
    S101_M_3_축3_전진_보조 AT %MW1104.1 : BOOL;
    S101_M_3_축3_전진단 AT %MW1104.3 : BOOL;
    S101_M_3_축3_조건 AT %MW1104.0 : BOOL;
    S101_M_3_축3_후진_LS_이상 AT %MW1104.6 : BOOL;
    S101_M_3_축3_후진_보조 AT %MW1104.2 : BOOL;
    S101_M_3_축3_후진단 AT %MW1104.4 : BOOL;
    S101_M_3축로보트_CTR_통신이상 AT %MW1024.8 : BOOL;
    S101_M_3축로보트_FRT_통신이상 AT %MW1024.7 : BOOL;
    S101_M_3축로보트_RR_통신이상 AT %MW1024.9 : BOOL;
    S101_M_ACT_선택_1 AT %MW1040.0 : BOOL;
    S101_M_ACT_선택_10 AT %MW1040.9 : BOOL;
    S101_M_ACT_선택_11 AT %MW1040.10 : BOOL;
    S101_M_ACT_선택_12 AT %MW1040.11 : BOOL;
    S101_M_ACT_선택_13 AT %MW1040.12 : BOOL;
    S101_M_ACT_선택_14 AT %MW1040.13 : BOOL;
    S101_M_ACT_선택_15 AT %MW1040.14 : BOOL;
    S101_M_ACT_선택_16 AT %MW1040.15 : BOOL;
    S101_M_ACT_선택_17 AT %MW1041.0 : BOOL;
    S101_M_ACT_선택_18 AT %MW1041.1 : BOOL;
    S101_M_ACT_선택_19 AT %MW1041.2 : BOOL;
    S101_M_ACT_선택_2 AT %MW1040.1 : BOOL;
    S101_M_ACT_선택_20 AT %MW1041.3 : BOOL;
    S101_M_ACT_선택_21 AT %MW1041.4 : BOOL;
    S101_M_ACT_선택_22 AT %MW1041.5 : BOOL;
    S101_M_ACT_선택_23 AT %MW1041.6 : BOOL;
    S101_M_ACT_선택_24 AT %MW1041.7 : BOOL;
    S101_M_ACT_선택_25 AT %MW1041.8 : BOOL;
    S101_M_ACT_선택_26 AT %MW1041.9 : BOOL;
    S101_M_ACT_선택_27 AT %MW1041.10 : BOOL;
    S101_M_ACT_선택_28 AT %MW1041.11 : BOOL;
    S101_M_ACT_선택_29 AT %MW1041.12 : BOOL;
    S101_M_ACT_선택_3 AT %MW1040.2 : BOOL;
    S101_M_ACT_선택_30 AT %MW1041.13 : BOOL;
    S101_M_ACT_선택_31 AT %MW1041.14 : BOOL;
    S101_M_ACT_선택_32 AT %MW1041.15 : BOOL;
    S101_M_ACT_선택_4 AT %MW1040.3 : BOOL;
    S101_M_ACT_선택_5 AT %MW1040.4 : BOOL;
    S101_M_ACT_선택_6 AT %MW1040.5 : BOOL;
    S101_M_ACT_선택_7 AT %MW1040.6 : BOOL;
    S101_M_ACT_선택_8 AT %MW1040.7 : BOOL;
    S101_M_ACT_선택_9 AT %MW1040.8 : BOOL;
    S101_M_APRON_LH_안착OK_POS AT %MW1004.8 : BOOL;
    S101_M_APRON_LH_제품감지_이상 AT %MW1014.0 : BOOL;
    S101_M_APRON_RH_안착OK_POS AT %MW1004.9 : BOOL;
    S101_M_APRON_RH_제품감지_이상 AT %MW1014.1 : BOOL;
    S101_M_APRON_랙방1_2_통신이상 AT %MW1024.1 : BOOL;
    S101_M_APRON_랙방3_4_통신이상 AT %MW1024.2 : BOOL;
    S101_M_APR_LH_사양_이상 AT %MW1016.0 : BOOL;
    S101_M_APR_RH_사양_이상 AT %MW1016.1 : BOOL;
    S101_M_AX_래치_전진_LAMP AT %MW11100 : WORD;
    S101_M_AX_래치_전진_LS_이상 AT %MW1100.5 : BOOL;
    S101_M_AX_래치_전진_보조 AT %MW1100.1 : BOOL;
    S101_M_AX_래치_전진단 AT %MW1100.3 : BOOL;
    S101_M_AX_래치_조건 AT %MW1100.0 : BOOL;
    S101_M_AX_래치_후진_LAMP AT %MW11101 : WORD;
    S101_M_AX_래치_후진_LS_이상 AT %MW1100.6 : BOOL;
    S101_M_AX_래치_후진_보조 AT %MW1100.2 : BOOL;
    S101_M_AX_래치_후진단 AT %MW1100.4 : BOOL;
    S101_M_CTIME_OVER_ALRAM AT %MW1006.14 : BOOL;
    S101_M_CTIME_OVER_MUTE AT %MW1006.13 : BOOL;
    S101_M_DASH_사양_이상 AT %MW1016.2 : BOOL;
    S101_M_DASH_안착OK_POS AT %MW1004.10 : BOOL;
    S101_M_DASH_제품감지_이상 AT %MW1014.2 : BOOL;
    S101_M_DASH_클램프_전진_LAMP AT %MW11104 : WORD;
    S101_M_DASH_클램프_전진_LS_이상 AT %MW1105.5 : BOOL;
    S101_M_DASH_클램프_전진_보조 AT %MW1105.1 : BOOL;
    S101_M_DASH_클램프_전진단 AT %MW1105.3 : BOOL;
    S101_M_DASH_클램프_조건 AT %MW1105.0 : BOOL;
    S101_M_DASH_클램프_후진_LAMP AT %MW11105 : WORD;
    S101_M_DASH_클램프_후진_LS_이상 AT %MW1105.6 : BOOL;
    S101_M_DASH_클램프_후진_보조 AT %MW1105.2 : BOOL;
    S101_M_DASH_클램프_후진단 AT %MW1105.4 : BOOL;
    S101_M_DATA_삭제_PLS AT %MW9001.0 : BOOL; (* S101_M_DATA_삭제_PLS *)
    S101_M_DATA_삭제_SIGN AT %MW9001.1 : BOOL; (* S101_M_DATA_삭제_SIGN *)
    S101_M_DATA_삭제_완료 AT %MW9001.2 : BOOL; (* S101_M_DATA_삭제_완료 *)
    S101_M_DATA_전송_MEMO AT %MW9001.8 : BOOL; (* S101_M_DATA_전송_MEMO *)
    S101_M_DATA_전송_PLS AT %MW9001.9 : BOOL; (* S101_M_DATA_전송_PLS *)
    S101_M_DATA_전송_SIGN AT %MW9001.10 : BOOL; (* S101_M_DATA_전송_SIGN *)
    S101_M_DATA_전송_완료 AT %MW9001.11 : BOOL; (* S101_M_DATA_전송_완료 *)
    S101_M_FRT_취출OK_POS AT %MW1004.11 : BOOL;
    S101_M_GATE_DOOR_NORMAL AT %MW1006.4 : BOOL;
    S101_M_GATE_ESTOP_NORMAR AT %MW1006.3 : BOOL;
    S101_M_OP_ESTOP_NORMAL AT %MW1006.1 : BOOL;
    S101_M_R101_1_CN_MATCH_OK AT %MW1005.0 : BOOL;
    S101_M_R101_1_CT_MATCH_OK AT %MW1005.1 : BOOL;
    S101_M_R102_1_CN_MATCH_OK AT %MW1005.2 : BOOL;
    S101_M_R102_1_CT_MATCH_OK AT %MW1005.3 : BOOL;
    S101_M_RB_ESTOP_NORMAL AT %MW1006.2 : BOOL;
    S101_M_SAFTY_NO_INT AT %MW1004.4 : BOOL;
    S101_M_SEMI_자동_모드 AT %MW1000.2 : BOOL;
    S101_M_SEQ AT %MW10020 : WORD; (* S101_M_SEQ *)
    S101_M_SHIFT_전진_LAMP AT %MW11102 : WORD;
    S101_M_SHIFT_전진_LS_이상 AT %MW1101.5 : BOOL;
    S101_M_SHIFT_전진_보조 AT %MW1101.1 : BOOL;
    S101_M_SHIFT_전진단 AT %MW1101.3 : BOOL;
    S101_M_SHIFT_조건 AT %MW1101.0 : BOOL;
    S101_M_SHIFT_후진_LAMP AT %MW11103 : WORD;
    S101_M_SHIFT_후진_LS_이상 AT %MW1101.6 : BOOL;
    S101_M_SHIFT_후진_보조 AT %MW1101.2 : BOOL;
    S101_M_SHIFT_후진단 AT %MW1101.4 : BOOL;
    S101_M_SRV1_CP_OFF AT %MW1017.0 : BOOL;
    S101_M_SRV1_MC_이상 AT %MW1023.0 : BOOL;
    S101_M_SRV1_오버런 AT %MW1022.0 : BOOL;
    S101_M_SRV1_이상 AT %MW1020.0 : BOOL;
    S101_M_SRV2_CP_OFF AT %MW1017.1 : BOOL;
    S101_M_SRV2_MC_이상 AT %MW1023.1 : BOOL;
    S101_M_SRV2_오버런 AT %MW1022.1 : BOOL;
    S101_M_SRV2_이상 AT %MW1020.1 : BOOL;
    S101_M_SRV3_CP_OFF AT %MW1017.2 : BOOL;
    S101_M_SRV3_MC_이상 AT %MW1023.2 : BOOL;
    S101_M_SRV3_오버런 AT %MW1022.2 : BOOL;
    S101_M_SRV3_이상 AT %MW1020.2 : BOOL;
    S101_M_STN_DASH_로딩완료 AT %MW1001.12 : BOOL;
    S101_M_STN_FRT_FLR_취출완료 AT %MW1001.13 : BOOL;
    S101_M_STN_LH_로딩완료 AT %MW1001.10 : BOOL;
    S101_M_STN_RH_로딩완료 AT %MW1001.11 : BOOL;
    S101_M_STN_차종_NONE AT %MW1002.1 : BOOL;
    S101_M_STN_차종_ON AT %MW1002.0 : BOOL;
    S101_M_VIN_NO_1_2 AT %MW10031 : WORD; (* S101_M_VIN_NO_1_2 *)
    S101_M_VIN_NO_3_4 AT %MW10032 : WORD; (* S101_M_VIN_NO_3_4 *)
    S101_M_VIN_NO_5_6 AT %MW10033 : WORD; (* S101_M_VIN_NO_5_6 *)
    S101_M_VIN_NO_7_8 AT %MW10034 : WORD; (* S101_M_VIN_NO_7_8 *)
    S101_M_VIN_NO_9_10 AT %MW10035 : WORD; (* S101_M_VIN_NO_9_10 *)
    S101_M_공기압_이상 AT %MW1013.0 : BOOL;
    S101_M_공정_APRON_제품감지_OFF AT %MW1001.4 : BOOL;
    S101_M_공정_APRON_제품감지_ON AT %MW1001.3 : BOOL;
    S101_M_공정_DASH_제품감지_OFF AT %MW1001.6 : BOOL;
    S101_M_공정_DASH_제품감지_ON AT %MW1001.5 : BOOL;
    S101_M_공정_HOME_POSI AT %MW1004.0 : BOOL;
    S101_M_공정_SAFETY_NORMAL AT %MW1006.7 : BOOL;
    S101_M_공정_간섭무 AT %MW1004.1 : BOOL;
    S101_M_공정_사양감지_OK AT %MW1001.7 : BOOL;
    S101_M_공정_통신이상 AT %MW1024.0 : BOOL;
    S101_M_부저_정지_보조 AT %MW1000.11 : BOOL;
    S101_M_사양이상 AT %MW1019.0 : BOOL;
    S101_M_서보1_통신이상 AT %MW1024.4 : BOOL;
    S101_M_서보2_통신이상 AT %MW1024.5 : BOOL;
    S101_M_서보3_통신이상 AT %MW1024.6 : BOOL;
    S101_M_서보판넬_통신이상 AT %MW1024.3 : BOOL;
    S101_M_수동_모드 AT %MW1000.3 : BOOL;
    S101_M_운전준비_ON AT %MW1000.0 : BOOL;
    S101_M_이상_리셋_보조 AT %MW1000.10 : BOOL;
    S101_M_자동_START AT %MW1000.5 : BOOL;
    S101_M_자동_모드 AT %MW1000.1 : BOOL;
    S101_M_자동_운전중 AT %MW1000.4 : BOOL;
    S101_M_작업_완료 AT %MW1001.0 : BOOL;
    S101_M_작업_완료_보조 AT %MW1000.9 : BOOL;
    S101_M_전체_3축_로봇1차_작업완료 AT %MW1001.1 : BOOL;
    S101_M_전체_용접로보트_1차_작업완료 AT %MW1001.8 : BOOL;
    S101_M_전체_용접로보트_최종_작업완료 AT %MW1001.9 : BOOL;
    S101_M_전체_용접완료 AT %MW1011.0 : BOOL;
    S101_M_전체_클램프_잠김단 AT %MW1004.12 : BOOL;
    S101_M_차종1_AX AT %MW10021.0 : BOOL; (* S101_M_차종1_AX *)
    S101_M_차종1_B AT %MW10021.1 : BOOL; (* S101_M_차종1_B *)
    S101_M_차종1_C AT %MW10021.2 : BOOL; (* S101_M_차종1_C *)
    S101_M_차종1_D AT %MW10021.3 : BOOL; (* S101_M_차종1_D *)
    S101_M_차종1_E AT %MW10021.4 : BOOL; (* S101_M_차종1_E *)
    S101_M_차종1_F AT %MW10021.5 : BOOL; (* S101_M_차종1_F *)
    S101_M_차종1_G AT %MW10021.6 : BOOL; (* S101_M_차종1_G *)
    S101_M_차종1_H AT %MW10021.7 : BOOL; (* S101_M_차종1_H *)
    S101_M_차종2_3DR AT %MW10021.8 : BOOL; (* S101_M_차종2_3DR *)
    S101_M_차종2_4DR AT %MW10021.9 : BOOL; (* S101_M_차종2_4DR *)
    S101_M_차종2_5DR AT %MW10021.10 : BOOL; (* S101_M_차종2_5DR *)
    S101_M_차종2_SP1 AT %MW10021.12 : BOOL; (* S101_M_차종2_SP1 *)
    S101_M_차종2_SP2 AT %MW10021.13 : BOOL; (* S101_M_차종2_SP2 *)
    S101_M_차종2_WGN AT %MW10021.11 : BOOL; (* S101_M_차종2_WGN *)
    S101_M_차종3_LHD AT %MW10021.14 : BOOL; (* S101_M_차종3_LHD *)
    S101_M_차종3_RHD AT %MW10021.15 : BOOL; (* S101_M_차종3_RHD *)
    S101_M_차종4_EEC AT %MW10022.3 : BOOL; (* S101_M_차종4_EEC *)
    S101_M_차종4_SP1 AT %MW10022.8 : BOOL; (* S101_M_차종4_SP1 *)
    S101_M_차종4_SP2 AT %MW10022.9 : BOOL; (* S101_M_차종4_SP2 *)
    S101_M_차종4_SP3 AT %MW10022.11 : BOOL; (* S101_M_차종4_SP3 *)
    S101_M_차종4_SP4 AT %MW10022.12 : BOOL; (* S101_M_차종4_SP4 *)
    S101_M_차종4_SP5 AT %MW10022.13 : BOOL; (* S101_M_차종4_SP5 *)
    S101_M_차종4_SP6 AT %MW10022.14 : BOOL; (* S101_M_차종4_SP6 *)
    S101_M_차종4_SP7 AT %MW10022.15 : BOOL; (* S101_M_차종4_SP7 *)
    S101_M_차종4_내수 AT %MW10022.0 : BOOL; (* S101_M_차종4_내수 *)
    S101_M_차종4_러시아 AT %MW10022.10 : BOOL; (* S101_M_차종4_러시아 *)
    S101_M_차종4_북미 AT %MW10022.2 : BOOL; (* S101_M_차종4_북미 *)
    S101_M_차종4_브라질 AT %MW10022.7 : BOOL; (* S101_M_차종4_브라질 *)
    S101_M_차종4_수출 AT %MW10022.1 : BOOL; (* S101_M_차종4_수출 *)
    S101_M_차종4_중국 AT %MW10022.6 : BOOL; (* S101_M_차종4_중국 *)
    S101_M_차종4_중동 AT %MW10022.5 : BOOL; (* S101_M_차종4_중동 *)
    S101_M_차종4_호주 AT %MW10022.4 : BOOL; (* S101_M_차종4_호주 *)
    S101_M_차종5_AT AT %MW10023.1 : BOOL; (* S101_M_차종5_AT *)
    S101_M_차종5_MT AT %MW10023.0 : BOOL; (* S101_M_차종5_MT *)
    S101_M_차종5_SP1 AT %MW10023.2 : BOOL; (* S101_M_차종5_SP1 *)
    S101_M_차종6_DSROOF AT %MW10023.6 : BOOL; (* S101_M_차종6_DSROOF *)
    S101_M_차종6_SP1 AT %MW10023.7 : BOOL; (* S101_M_차종6_SP1 *)
    S101_M_차종6_썬루프 AT %MW10023.4 : BOOL; (* S101_M_차종6_썬루프 *)
    S101_M_차종6_일반루프 AT %MW10023.3 : BOOL; (* S101_M_차종6_일반루프 *)
    S101_M_차종6_파노라마루프 AT %MW10023.5 : BOOL; (* S101_M_차종6_파노라마루프 *)
    S101_M_차종7_DSL AT %MW10023.9 : BOOL; (* S101_M_차종7_DSL *)
    S101_M_차종7_GSL AT %MW10023.8 : BOOL; (* S101_M_차종7_GSL *)
    S101_M_차종7_SP1 AT %MW10023.10 : BOOL; (* S101_M_차종7_SP1 *)
    S101_M_차종7_SP2 AT %MW10023.11 : BOOL; (* S101_M_차종7_SP2 *)
    S101_M_차종7_SP3 AT %MW10023.12 : BOOL; (* S101_M_차종7_SP3 *)
    S101_M_차종7_SP4 AT %MW10023.13 : BOOL; (* S101_M_차종7_SP4 *)
    S101_M_차종7_SP5 AT %MW10023.14 : BOOL; (* S101_M_차종7_SP5 *)
    S101_M_차종7_SP6 AT %MW10023.15 : BOOL; (* S101_M_차종7_SP6 *)
    S101_M_차종8_2WD AT %MW10024.0 : BOOL; (* S101_M_차종8_2WD *)
    S101_M_차종8_4WD AT %MW10024.1 : BOOL; (* S101_M_차종8_4WD *)
    S101_M_차종8_SP1 AT %MW10024.2 : BOOL; (* S101_M_차종8_SP1 *)
    S101_M_차종9_MPI AT %MW10024.3 : BOOL; (* S101_M_차종9_MPI *)
    S101_M_차종9_SP1 AT %MW10024.5 : BOOL; (* S101_M_차종9_SP1 *)
    S101_M_차종9_SP10 AT %MW10024.14 : BOOL; (* S101_M_차종9_SP10 *)
    S101_M_차종9_SP11 AT %MW10024.15 : BOOL; (* S101_M_차종9_SP11 *)
    S101_M_차종9_SP2 AT %MW10024.6 : BOOL; (* S101_M_차종9_SP2 *)
    S101_M_차종9_SP3 AT %MW10024.7 : BOOL; (* S101_M_차종9_SP3 *)
    S101_M_차종9_SP4 AT %MW10024.8 : BOOL; (* S101_M_차종9_SP4 *)
    S101_M_차종9_SP5 AT %MW10024.9 : BOOL; (* S101_M_차종9_SP5 *)
    S101_M_차종9_SP6 AT %MW10024.10 : BOOL; (* S101_M_차종9_SP6 *)
    S101_M_차종9_SP7 AT %MW10024.11 : BOOL; (* S101_M_차종9_SP7 *)
    S101_M_차종9_SP8 AT %MW10024.12 : BOOL; (* S101_M_차종9_SP8 *)
    S101_M_차종9_SP9 AT %MW10024.13 : BOOL; (* S101_M_차종9_SP9 *)
    S101_M_차종9_T_GDI AT %MW10024.4 : BOOL; (* S101_M_차종9_T_GDI *)
    S101_M_차종_AS AT %MW10030.9 : BOOL; (* S101_M_차종_AS *)
    S101_M_차종_OPT1_R_RACK_무 AT %MW10025.3 : BOOL; (* S101_M_차종_OPT1_R_RACK_무 *)
    S101_M_차종_OPT1_R_RACK_유 AT %MW10025.2 : BOOL; (* S101_M_차종_OPT1_R_RACK_유 *)
    S101_M_차종_OPT1_SP1 AT %MW10025.10 : BOOL; (* S101_M_차종_OPT1_SP1 *)
    S101_M_차종_OPT1_SP2 AT %MW10025.11 : BOOL; (* S101_M_차종_OPT1_SP2 *)
    S101_M_차종_OPT1_SP3 AT %MW10025.12 : BOOL; (* S101_M_차종_OPT1_SP3 *)
    S101_M_차종_OPT1_SP4 AT %MW10025.13 : BOOL; (* S101_M_차종_OPT1_SP4 *)
    S101_M_차종_OPT1_SP5 AT %MW10025.14 : BOOL; (* S101_M_차종_OPT1_SP5 *)
    S101_M_차종_OPT1_SP6 AT %MW10025.15 : BOOL; (* S101_M_차종_OPT1_SP6 *)
    S101_M_차종_OPT1_S_REP_EATER_무 AT %MW10025.7 : BOOL; (* S101_M_차종_OPT1_S_REP_EATER_무 *)
    S101_M_차종_OPT1_S_REP_EATER_유 AT %MW10025.6 : BOOL; (* S101_M_차종_OPT1_S_REP_EATER_유 *)
    S101_M_차종_OPT1_VAN_무 AT %MW10025.9 : BOOL; (* S101_M_차종_OPT1_VAN_무 *)
    S101_M_차종_OPT1_VAN_유 AT %MW10025.8 : BOOL; (* S101_M_차종_OPT1_VAN_유 *)
    S101_M_차종_OPT1_슬라이딩_무 AT %MW10025.1 : BOOL; (* S101_M_차종_OPT1_슬라이딩_무 *)
    S101_M_차종_OPT1_슬라이딩_유 AT %MW10025.0 : BOOL; (* S101_M_차종_OPT1_슬라이딩_유 *)
    S101_M_차종_OPT1_폴딩_무 AT %MW10025.5 : BOOL; (* S101_M_차종_OPT1_폴딩_무 *)
    S101_M_차종_OPT1_폴딩_유 AT %MW10025.4 : BOOL; (* S101_M_차종_OPT1_폴딩_유 *)
    S101_M_차종_OPT2_SP_WORD1 AT %MW10026 : WORD; (* S101_M_차종_OPT2_SP_WORD1 *)
    S101_M_차종_OPT3_SP_WORD2 AT %MW10027 : WORD; (* S101_M_차종_OPT3_SP_WORD2 *)
    S101_M_차종_OPT4_SP_WORD3 AT %MW10028 : WORD; (* S101_M_차종_OPT4_SP_WORD3 *)
    S101_M_차종_OPT5_SP_WORD4 AT %MW10029 : WORD; (* S101_M_차종_OPT5_SP_WORD4 *)
    S101_M_차종_SP1 AT %MW10030.0 : BOOL; (* S101_M_차종_SP1 *)
    S101_M_차종_SP2 AT %MW10030.1 : BOOL; (* S101_M_차종_SP2 *)
    S101_M_차종_SP3 AT %MW10030.2 : BOOL; (* S101_M_차종_SP3 *)
    S101_M_차종_SP4 AT %MW10030.3 : BOOL; (* S101_M_차종_SP4 *)
    S101_M_차종_SP5 AT %MW10030.4 : BOOL; (* S101_M_차종_SP5 *)
    S101_M_차종_SP6 AT %MW10030.5 : BOOL; (* S101_M_차종_SP6 *)
    S101_M_차종_SP7 AT %MW10030.6 : BOOL; (* S101_M_차종_SP7 *)
    S101_M_차종_SP8 AT %MW10030.7 : BOOL; (* S101_M_차종_SP8 *)
    S101_M_차종_SP9 AT %MW10030.15 : BOOL; (* S101_M_차종_SP9 *)
    S101_M_차종_공대차 AT %MW10030.12 : BOOL; (* S101_M_차종_공대차 *)
    S101_M_차종_공차 AT %MW10030.10 : BOOL; (* S101_M_차종_공차 *)
    S101_M_차종_불량대차 AT %MW10030.13 : BOOL; (* S101_M_차종_불량대차 *)
    S101_M_차종_불량차 AT %MW10030.11 : BOOL; (* S101_M_차종_불량차 *)
    S101_M_차종_비축 AT %MW10030.8 : BOOL; (* S101_M_차종_비축 *)
    S101_M_차종_이상 AT %MW1015.2 : BOOL;
    S101_M_차종_취출대차 AT %MW10030.14 : BOOL; (* S101_M_차종_취출대차 *)
